LIN {X 0,Y 428.586,Z 1043.755,A -85,B 0,C 180,E1 19403.227,E2 19403.227} C_VEL
LIN {X 0,Y 431.846,Z 1036.608,A -85,B 0,C 180,E1 19403.942,E2 19403.942} C_VEL
LIN {X 0,Y 434.974,Z 1024.331,A -85,B 0,C 180,E1 19405.544,E2 19405.544} C_VEL
LIN {X 0,Y 437.859,Z 1011.623,A -85,B 0,C 180,E1 19407.088,E2 19407.088} C_VEL
LIN {X 0,Y 455.696,Z 965.576,A -85,B 0,C 180,E1 19410.268,E2 19410.268} C_VEL
LIN {X 0,Y 463.791,Z 940.685,A -85,B 0,C 180,E1 19411.605,E2 19411.605} C_VEL
LIN {X 0,Y 457.575,Z 919.275,A -85,B 0,C 180,E1 19415.61,E2 19415.61} C_VEL
LIN {X 0,Y 449.958,Z 899.264,A -85,B 0,C 180,E1 19420.368,E2 19420.368} C_VEL
LIN {X 0,Y 443.441,Z 884.682,A -85,B 0,C 180,E1 19425.003,E2 19425.003} C_VEL
LIN {X 0,Y 438.178,Z 874.111,A -85,B 0,C 180,E1 19429.684,E2 19429.684} C_VEL
LIN {X 0,Y 435.63,Z 868.79,A -85,B 0,C 180,E1 19433.016,E2 19433.016} C_VEL
LIN {X 0,Y 433.736,Z 862.951,A -85,B 0,C 180,E1 19438.99,E2 19438.99} C_VEL
LIN {X 0,Y 433.685,Z 863.847,A -85,B 0,C 180,E1 19442.859,E2 19442.859} C_VEL
LIN {X 0,Y 435.972,Z 870.801,A -85,B 0,C 180,E1 19448.898,E2 19448.898} C_VEL
LIN {X 0,Y 440.304,Z 880.375,A -85,B 0,C 180,E1 19453.887,E2 19453.887} C_VEL
LIN {X 0,Y 447.364,Z 897.231,A -85,B 0,C 180,E1 19459.727,E2 19459.727} C_VEL
LIN {X 0,Y 454.424,Z 917.787,A -85,B 0,C 180,E1 19464.863,E2 19464.863} C_VEL
LIN {X 0,Y 460.195,Z 940.594,A -85,B 0,C 180,E1 19469.353,E2 19469.353} C_VEL
LIN {X 0,Y 444.53,Z 983.942,A -85,B 0,C 180,E1 19472.239,E2 19472.239} C_VEL
LIN {X 0,Y 426.136,Z 1025.719,A -85,B 0,C 180,E1 19476.025,E2 19476.025} C_VEL
LIN {X 0,Y 408.075,Z 1061.829,A -85,B 0,C 180,E1 19480.461,E2 19480.461} C_VEL
LIN {X 0,Y 389.858,Z 1095.549,A -85,B 0,C 180,E1 19486.146,E2 19486.146} C_VEL
LIN {X 0,Y 374.87,Z 1122.588,A -85,B 0,C 180,E1 19492.358,E2 19492.358} C_VEL
LIN {X 0,Y 362.214,Z 1146.532,A -85,B 0,C 180,E1 19499.96,E2 19499.96} C_VEL
LIN {X 0,Y 354.663,Z 1163.186,A -85,B 0,C 180,E1 19507.453,E2 19507.453} C_VEL
LIN {X 0,Y 350.741,Z 1174.594,A -85,B 0,C 180,E1 19515.02,E2 19515.02} C_VEL
LIN {X 0,Y 349.218,Z 1181.313,A -85,B 0,C 180,E1 19522.542,E2 19522.542} C_VEL
LIN {X 0,Y 349.207,Z 1183.553,A -85,B 0,C 180,E1 19530.001,E2 19530.001} C_VEL
LIN {X 0,Y 349.289,Z 1181.244,A -85,B 0,C 180,E1 19537.459,E2 19537.459} C_VEL
LIN {X 0,Y 350.779,Z 1174.475,A -85,B 0,C 180,E1 19544.981,E2 19544.981} C_VEL
LIN {X 0,Y 354.739,Z 1163.013,A -85,B 0,C 180,E1 19552.545,E2 19552.545} C_VEL
LIN {X 0,Y 362.329,Z 1146.279,A -85,B 0,C 180,E1 19560.032,E2 19560.032} C_VEL
LIN {X 0,Y 375.056,Z 1122.213,A -85,B 0,C 180,E1 19567.648,E2 19567.648} C_VEL
LIN {X 0,Y 390.041,Z 1095.14,A -85,B 0,C 180,E1 19573.831,E2 19573.831} C_VEL
LIN {X 0,Y 408.55,Z 1060.855,A -85,B 0,C 180,E1 19579.582,E2 19579.582} C_VEL
LIN {X 0,Y 426.873,Z 1023.878,A -85,B 0,C 180,E1 19584.075,E2 19584.075} C_VEL
LIN {X 0,Y 444.921,Z 983.008,A -85,B 0,C 180,E1 19587.716,E2 19587.716} C_VEL
LIN {X 0,Y 460.201,Z 940.721,A -85,B 0,C 180,E1 19590.509,E2 19590.509} C_VEL
LIN {X 0,Y 454.389,Z 918.018,A -85,B 0,C 180,E1 19594.981,E2 19594.981} C_VEL
LIN {X 0,Y 447.112,Z 896.88,A -85,B 0,C 180,E1 19600.261,E2 19600.261} C_VEL
LIN {X 0,Y 440.513,Z 881.043,A -85,B 0,C 180,E1 19605.668,E2 19605.668} C_VEL
LIN {X 0,Y 436.198,Z 871.856,A -85,B 0,C 180,E1 19610.353,E2 19610.353} C_VEL
LIN {X 0,Y 434.863,Z 868.474,A -85,B 0,C 180,E1 19612.525,E2 19612.525} C_VEL
LIN {X 0,Y 433.446,Z 862.89,A -85,B 0,C 180,E1 19618.014,E2 19618.014} C_VEL
LIN {X 0,Y 433.74,Z 863.748,A -85,B 0,C 180,E1 19622.632,E2 19622.632} C_VEL
LIN {X 0,Y 436.694,Z 870.999,A -85,B 0,C 180,E1 19628.718,E2 19628.718} C_VEL
LIN {X 0,Y 441.953,Z 881.235,A -85,B 0,C 180,E1 19633.858,E2 19633.858} C_VEL
LIN {X 0,Y 449.143,Z 897.26,A -85,B 0,C 180,E1 19639.159,E2 19639.159} C_VEL
LIN {X 0,Y 457.134,Z 917.905,A -85,B 0,C 180,E1 19644.155,E2 19644.155} C_VEL
LIN {X 0,Y 463.866,Z 940.396,A -85,B 0,C 180,E1 19648.408,E2 19648.408} C_VEL
LIN {X 0,Y 449.596,Z 982.266,A -85,B 0,C 180,E1 19650.775,E2 19650.775} C_VEL
LIN {X 0,Y 431.875,Z 1025.293,A -85,B 0,C 180,E1 19654.114,E2 19654.114} C_VEL
LIN {X 0,Y 413.975,Z 1063.618,A -85,B 0,C 180,E1 19658.166,E2 19658.166} C_VEL
LIN {X 0,Y 395.325,Z 1100.234,A -85,B 0,C 180,E1 19663.486,E2 19663.486} C_VEL
LIN {X 0,Y 379.922,Z 1129.531,A -85,B 0,C 180,E1 19669.197,E2 19669.197} C_VEL
LIN {X 0,Y 366.111,Z 1156.35,A -85,B 0,C 180,E1 19676.315,E2 19676.315} C_VEL
LIN {X 0,Y 357.094,Z 1176.529,A -85,B 0,C 180,E1 19683.618,E2 19683.618} C_VEL
LIN {X 0,Y 351.628,Z 1191.995,A -85,B 0,C 180,E1 19691.651,E2 19691.651} C_VEL
LIN {X 0,Y 349.589,Z 1200.987,A -85,B 0,C 180,E1 19698.782,E2 19698.782} C_VEL
LIN {X 0,Y 349.086,Z 1205.302,A -85,B 0,C 180,E1 19705.032,E2 19705.032} C_VEL
LIN {X 0,Y 349.253,Z 1206.48,A -85,B 0,C 180,E1 19709.999,E2 19709.999} C_VEL
LIN {X 0,Y 349.173,Z 1204.011,A -85,B 0,C 180,E1 19717.459,E2 19717.459} C_VEL
LIN {X 0,Y 350.156,Z 1197.853,A -85,B 0,C 180,E1 19724.149,E2 19724.149} C_VEL
LIN {X 0,Y 353.578,Z 1185.77,A -85,B 0,C 180,E1 19731.958,E2 19731.958} C_VEL
LIN {X 0,Y 360.388,Z 1168.719,A -85,B 0,C 180,E1 19739.515,E2 19739.515} C_VEL
LIN {X 0,Y 372.131,Z 1144.328,A -85,B 0,C 180,E1 19747.157,E2 19747.157} C_VEL
LIN {X 0,Y 387.149,Z 1115.813,A -85,B 0,C 180,E1 19753.702,E2 19753.702} C_VEL
LIN {X 0,Y 405.824,Z 1080.003,A -85,B 0,C 180,E1 19759.666,E2 19759.666} C_VEL
LIN {X 0,Y 423.714,Z 1043.487,A -85,B 0,C 180,E1 19764.118,E2 19764.118} C_VEL
LIN {X 0,Y 437.859,Z 1011.623,A -85,B 0,C 180,E1 19767.088,E2 19767.088} C_VEL
LIN {X 0,Y 443.734,Z 986.824,A -85,B 0,C 180,E1 19769.787,E2 19769.787} C_VEL
LIN {X 0,Y 444.408,Z 984.999,A -85,B 0,C 180,E1 19769.923,E2 19769.923} C_VEL
LIN {X 0,Y 458.785,Z 943.642,A -85,B 0,C 180,E1 19772.398,E2 19772.398} C_VEL
LIN {X 0,Y 451.781,Z 920.233,A -85,B 0,C 180,E1 19777.109,E2 19777.109} C_VEL
LIN {X 0,Y 444.419,Z 900.847,A -85,B 0,C 180,E1 19782.183,E2 19782.183} C_VEL
LIN {X 0,Y 438.462,Z 887.226,A -85,B 0,C 180,E1 19787.045,E2 19787.045} C_VEL
LIN {X 0,Y 434.775,Z 879.627,A -85,B 0,C 180,E1 19790.991,E2 19790.991} C_VEL
LIN {X 0,Y 433.267,Z 876.2,A -85,B 0,C 180,E1 19793.229,E2 19793.229} C_VEL
LIN {X 0,Y 431.551,Z 870.535,A -85,B 0,C 180,E1 19798.985,E2 19798.985} C_VEL
LIN {X 0,Y 431.475,Z 871.393,A -85,B 0,C 180,E1 19802.748,E2 19802.748} C_VEL
LIN {X 0,Y 433.507,Z 877.891,A -85,B 0,C 180,E1 19808.536,E2 19808.536} C_VEL
LIN {X 0,Y 437.705,Z 888.299,A -85,B 0,C 180,E1 19813.971,E2 19813.971} C_VEL
LIN {X 0,Y 443.762,Z 903.724,A -85,B 0,C 180,E1 19819.376,E2 19819.376} C_VEL
LIN {X 0,Y 450.263,Z 923.937,A -85,B 0,C 180,E1 19824.524,E2 19824.524} C_VEL
LIN {X 0,Y 455.052,Z 944.062,A -85,B 0,C 180,E1 19828.604,E2 19828.604} C_VEL
LIN {X 0,Y 443.783,Z 975.55,A -85,B 0,C 180,E1 19830.729,E2 19830.729} C_VEL
LIN {X 0,Y 426.406,Z 1015.666,A -85,B 0,C 180,E1 19834.07,E2 19834.07} C_VEL
LIN {X 0,Y 407.054,Z 1054.1,A -85,B 0,C 180,E1 19838.476,E2 19838.476} C_VEL
LIN {X 0,Y 388.95,Z 1087.233,A -85,B 0,C 180,E1 19843.65,E2 19843.65} C_VEL
LIN {X 0,Y 372.018,Z 1116.573,A -85,B 0,C 180,E1 19849.952,E2 19849.952} C_VEL
LIN {X 0,Y 358.903,Z 1140.024,A -85,B 0,C 180,E1 19856.816,E2 19856.816} C_VEL
LIN {X 0,Y 348.66,Z 1159.953,A -85,B 0,C 180,E1 19865.102,E2 19865.102} C_VEL
LIN {X 0,Y 344.049,Z 1171.621,A -85,B 0,C 180,E1 19872.096,E2 19872.096} C_VEL
LIN {X 0,Y 341.71,Z 1179.921,A -85,B 0,C 180,E1 19879.813,E2 19879.813} C_VEL
LIN {X 0,Y 341.121,Z 1183.502,A -85,B 0,C 180,E1 19887.462,E2 19887.462} C_VEL
LIN {X 0,Y 341.232,Z 1183.485,A -85,B 0,C 180,E1 19892.539,E2 19892.539} C_VEL
LIN {X 0,Y 341.765,Z 1179.847,A -85,B 0,C 180,E1 19900.188,E2 19900.188} C_VEL
LIN {X 0,Y 344.103,Z 1171.477,A -85,B 0,C 180,E1 19907.904,E2 19907.904} C_VEL
LIN {X 0,Y 350.078,Z 1156.974,A -85,B 0,C 180,E1 19916.261,E2 19916.261} C_VEL
LIN {X 0,Y 359.934,Z 1137.868,A -85,B 0,C 180,E1 19923.8,E2 19923.8} C_VEL
LIN {X 0,Y 374.138,Z 1112.783,A -85,B 0,C 180,E1 19930.895,E2 19930.895} C_VEL
LIN {X 0,Y 390.81,Z 1083.708,A -85,B 0,C 180,E1 19936.873,E2 19936.873} C_VEL
LIN {X 0,Y 409.721,Z 1049.044,A -85,B 0,C 180,E1 19942.082,E2 19942.082} C_VEL
LIN {X 0,Y 427.732,Z 1012.531,A -85,B 0,C 180,E1 19946.123,E2 19946.123} C_VEL
LIN {X 0,Y 446.584,Z 968.32,A -85,B 0,C 180,E1 19949.677,E2 19949.677} C_VEL
LIN {X 0,Y 455.082,Z 944.515,A -85,B 0,C 180,E1 19951.205,E2 19951.205} C_VEL
LIN {X 0,Y 449.389,Z 921.401,A -85,B 0,C 180,E1 19955.954,E2 19955.954} C_VEL
LIN {X 0,Y 442.896,Z 901.812,A -85,B 0,C 180,E1 19961.102,E2 19961.102} C_VEL
LIN {X 0,Y 437.485,Z 887.883,A -85,B 0,C 180,E1 19966.022,E2 19966.022} C_VEL
LIN {X 0,Y 432.894,Z 876.3,A -85,B 0,C 180,E1 19972.202,E2 19972.202} C_VEL
LIN {X 0,Y 431.26,Z 870.482,A -85,B 0,C 180,E1 19978.004,E2 19978.004} C_VEL
LIN {X 0,Y 431.52,Z 871.282,A -85,B 0,C 180,E1 19982.52,E2 19982.52} C_VEL
LIN {X 0,Y 434.321,Z 878.522,A -85,B 0,C 180,E1 19988.575,E2 19988.575} C_VEL
LIN {X 0,Y 438.944,Z 887.899,A -85,B 0,C 180,E1 19993.447,E2 19993.447} C_VEL
LIN {X 0,Y 445.778,Z 903.809,A -85,B 0,C 180,E1 19998.795,E2 19998.795} C_VEL
LIN {X 0,Y 453.312,Z 924.562,A -85,B 0,C 180,E1 20003.896,E2 20003.896} C_VEL
LIN {X 0,Y 458.761,Z 943.784,A -85,B 0,C 180,E1 20007.646,E2 20007.646} C_VEL
LIN {X 0,Y 442.236,Z 990.175,A -85,B 0,C 180,E1 20010.438,E2 20010.438} C_VEL
LIN {X 0,Y 424.86,Z 1030.734,A -85,B 0,C 180,E1 20013.733,E2 20013.733} C_VEL
LIN {X 0,Y 405.075,Z 1070.686,A -85,B 0,C 180,E1 20018.2,E2 20018.2} C_VEL
LIN {X 0,Y 386.799,Z 1105.278,A -85,B 0,C 180,E1 20023.515,E2 20023.515} C_VEL
LIN {X 0,Y 369.335,Z 1137.111,A -85,B 0,C 180,E1 20030.255,E2 20030.255} C_VEL
LIN {X 0,Y 356.233,Z 1162.098,A -85,B 0,C 180,E1 20037.567,E2 20037.567} C_VEL
LIN {X 0,Y 347.526,Z 1181.212,A -85,B 0,C 180,E1 20045.333,E2 20045.333} C_VEL
LIN {X 0,Y 343.523,Z 1193.016,A -85,B 0,C 180,E1 20052.065,E2 20052.065} C_VEL
LIN {X 0,Y 341.538,Z 1201.955,A -85,B 0,C 180,E1 20059.805,E2 20059.805} C_VEL
LIN {X 0,Y 341.228,Z 1205.87,A -85,B 0,C 180,E1 20067.461,E2 20067.461} C_VEL
LIN {X 0,Y 341.323,Z 1205.874,A -85,B 0,C 180,E1 20072.536,E2 20072.536} C_VEL
LIN {X 0,Y 341.534,Z 1201.962,A -85,B 0,C 180,E1 20080.193,E2 20080.193} C_VEL
LIN {X 0,Y 343.512,Z 1193.03,A -85,B 0,C 180,E1 20087.933,E2 20087.933} C_VEL
LIN {X 0,Y 348.459,Z 1179.029,A -85,B 0,C 180,E1 20095.698,E2 20095.698} C_VEL
LIN {X 0,Y 357.511,Z 1159.576,A -85,B 0,C 180,E1 20103.33,E2 20103.33} C_VEL
LIN {X 0,Y 371.226,Z 1133.502,A -85,B 0,C 180,E1 20110.638,E2 20110.638} C_VEL
LIN {X 0,Y 388.234,Z 1102.606,A -85,B 0,C 180,E1 20116.975,E2 20116.975} C_VEL
LIN {X 0,Y 408.129,Z 1064.976,A -85,B 0,C 180,E1 20122.545,E2 20122.545} C_VEL
LIN {X 0,Y 426.367,Z 1027.477,A -85,B 0,C 180,E1 20126.576,E2 20126.576} C_VEL
LIN {X 0,Y 444.095,Z 985.792,A -85,B 0,C 180,E1 20129.867,E2 20129.867} C_VEL
LIN {X 0,Y 444.408,Z 984.999,A -85,B 0,C 180,E1 20129.923,E2 20129.923} C_VEL
LIN {X 0,Y 447.634,Z 971.252,A -85,B 0,C 180,E1 20131.267,E2 20131.267} C_VEL
LIN {X 0,Y 450.696,Z 957.074,A -85,B 0,C 180,E1 20132.515,E2 20132.515} C_VEL
LIN {X 0,Y 453.804,Z 947.912,A -85,B 0,C 180,E1 20133.003,E2 20133.003} C_VEL
LIN {X 0,Y 447.279,Z 924.708,A -85,B 0,C 180,E1 20137.868,E2 20137.868} C_VEL
LIN {X 0,Y 440.411,Z 905.787,A -85,B 0,C 180,E1 20143.033,E2 20143.033} C_VEL
LIN {X 0,Y 434.032,Z 890.643,A -85,B 0,C 180,E1 20148.95,E2 20148.95} C_VEL
LIN {X 0,Y 430.496,Z 883.205,A -85,B 0,C 180,E1 20153.944,E2 20153.944} C_VEL
LIN {X 0,Y 429.364,Z 878.125,A -85,B 0,C 180,E1 20158.98,E2 20158.98} C_VEL
LIN {X 0,Y 429.347,Z 878.148,A -85,B 0,C 180,E1 20162.005,E2 20162.005} C_VEL
LIN {X 0,Y 430.92,Z 885.665,A -85,B 0,C 180,E1 20168.588,E2 20168.588} C_VEL
LIN {X 0,Y 435.081,Z 896.244,A -85,B 0,C 180,E1 20174.057,E2 20174.057} C_VEL
LIN {X 0,Y 440.747,Z 911.938,A -85,B 0,C 180,E1 20179.514,E2 20179.514} C_VEL
LIN {X 0,Y 446.572,Z 932.006,A -85,B 0,C 180,E1 20184.606,E2 20184.606} C_VEL
LIN {X 0,Y 450.102,Z 948.566,A -85,B 0,C 180,E1 20188.019,E2 20188.019} C_VEL
LIN {X 0,Y 431.793,Z 994.267,A -85,B 0,C 180,E1 20191.22,E2 20191.22} C_VEL
LIN {X 0,Y 413.229,Z 1033.294,A -85,B 0,C 180,E1 20194.973,E2 20194.973} C_VEL
LIN {X 0,Y 393.426,Z 1069.906,A -85,B 0,C 180,E1 20199.811,E2 20199.811} C_VEL
LIN {X 0,Y 375.588,Z 1100.457,A -85,B 0,C 180,E1 20205.308,E2 20205.308} C_VEL
LIN {X 0,Y 358.669,Z 1128.649,A -85,B 0,C 180,E1 20212.347,E2 20212.347} C_VEL
LIN {X 0,Y 347.218,Z 1148.728,A -85,B 0,C 180,E1 20219.247,E2 20219.247} C_VEL
LIN {X 0,Y 339.184,Z 1164.828,A -85,B 0,C 180,E1 20227.058,E2 20227.058} C_VEL
LIN {X 0,Y 335.205,Z 1175.121,A -85,B 0,C 180,E1 20234.308,E2 20234.308} C_VEL
LIN {X 0,Y 333.46,Z 1181.833,A -85,B 0,C 180,E1 20242.188,E2 20242.188} C_VEL
LIN {X 0,Y 333.411,Z 1184.071,A -85,B 0,C 180,E1 20250.001,E2 20250.001} C_VEL
LIN {X 0,Y 333.521,Z 1181.766,A -85,B 0,C 180,E1 20257.813,E2 20257.813} C_VEL
LIN {X 0,Y 335.256,Z 1175.005,A -85,B 0,C 180,E1 20265.692,E2 20265.692} C_VEL
LIN {X 0,Y 340.463,Z 1162.3,A -85,B 0,C 180,E1 20274.31,E2 20274.31} C_VEL
LIN {X 0,Y 350.146,Z 1143.453,A -85,B 0,C 180,E1 20282.641,E2 20282.641} C_VEL
LIN {X 0,Y 363.929,Z 1119.888,A -85,B 0,C 180,E1 20290.007,E2 20290.007} C_VEL
LIN {X 0,Y 381.77,Z 1089.961,A -85,B 0,C 180,E1 20296.663,E2 20296.663} C_VEL
LIN {X 0,Y 400.454,Z 1057.184,A -85,B 0,C 180,E1 20301.952,E2 20301.952} C_VEL
LIN {X 0,Y 420.938,Z 1017.603,A -85,B 0,C 180,E1 20306.581,E2 20306.581} C_VEL
LIN {X 0,Y 439.163,Z 977.032,A -85,B 0,C 180,E1 20309.977,E2 20309.977} C_VEL
LIN {X 0,Y 449.962,Z 948.025,A -85,B 0,C 180,E1 20311.972,E2 20311.972} C_VEL
LIN {X 0,Y 444.767,Z 925.808,A -85,B 0,C 180,E1 20316.718,E2 20316.718} C_VEL
LIN {X 0,Y 438.761,Z 906.785,A -85,B 0,C 180,E1 20321.957,E2 20321.957} C_VEL
LIN {X 0,Y 433.906,Z 893.651,A -85,B 0,C 180,E1 20326.931,E2 20326.931} C_VEL
LIN {X 0,Y 430.008,Z 883.44,A -85,B 0,C 180,E1 20332.812,E2 20332.812} C_VEL
LIN {X 0,Y 429.073,Z 878.075,A -85,B 0,C 180,E1 20337.994,E2 20337.994} C_VEL
LIN {X 0,Y 429.294,Z 879.012,A -85,B 0,C 180,E1 20342.533,E2 20342.533} C_VEL
LIN {X 0,Y 432.017,Z 886.651,A -85,B 0,C 180,E1 20348.81,E2 20348.81} C_VEL
LIN {X 0,Y 436.314,Z 895.901,A -85,B 0,C 180,E1 20353.53,E2 20353.53} C_VEL
LIN {X 0,Y 442.771,Z 912.014,A -85,B 0,C 180,E1 20358.928,E2 20358.928} C_VEL
LIN {X 0,Y 449.428,Z 931.869,A -85,B 0,C 180,E1 20363.805,E2 20363.805} C_VEL
LIN {X 0,Y 453.692,Z 947.9,A -85,B 0,C 180,E1 20367.002,E2 20367.002} C_VEL
LIN {X 0,Y 436.967,Z 992.903,A -85,B 0,C 180,E1 20369.729,E2 20369.729} C_VEL
LIN {X 0,Y 419.212,Z 1032.761,A -85,B 0,C 180,E1 20373.026,E2 20373.026} C_VEL
LIN {X 0,Y 398.464,Z 1073.371,A -85,B 0,C 180,E1 20377.658,E2 20377.658} C_VEL
LIN {X 0,Y 379.725,Z 1107.337,A -85,B 0,C 180,E1 20383.042,E2 20383.042} C_VEL
LIN {X 0,Y 362.274,Z 1138.074,A -85,B 0,C 180,E1 20389.718,E2 20389.718} C_VEL
LIN {X 0,Y 348.73,Z 1162.77,A -85,B 0,C 180,E1 20397.174,E2 20397.174} C_VEL
LIN {X 0,Y 339.719,Z 1181.772,A -85,B 0,C 180,E1 20405.153,E2 20405.153} C_VEL
LIN {X 0,Y 335.255,Z 1194.611,A -85,B 0,C 180,E1 20412.962,E2 20412.962} C_VEL
LIN {X 0,Y 333.664,Z 1201.692,A -85,B 0,C 180,E1 20419.562,E2 20419.562} C_VEL
LIN {X 0,Y 333.322,Z 1205.61,A -85,B 0,C 180,E1 20427.4,E2 20427.4} C_VEL
LIN {X 0,Y 333.413,Z 1205.614,A -85,B 0,C 180,E1 20432.596,E2 20432.596} C_VEL
LIN {X 0,Y 333.659,Z 1201.7,A -85,B 0,C 180,E1 20440.436,E2 20440.436} C_VEL
LIN {X 0,Y 335.787,Z 1192.764,A -85,B 0,C 180,E1 20448.36,E2 20448.36} C_VEL
LIN {X 0,Y 341.553,Z 1177.754,A -85,B 0,C 180,E1 20456.777,E2 20456.777} C_VEL
LIN {X 0,Y 351.226,Z 1158.109,A -85,B 0,C 180,E1 20464.458,E2 20464.458} C_VEL
LIN {X 0,Y 366.464,Z 1130.803,A -85,B 0,C 180,E1 20472.066,E2 20472.066} C_VEL
LIN {X 0,Y 383.468,Z 1100.772,A -85,B 0,C 180,E1 20478.15,E2 20478.15} C_VEL
LIN {X 0,Y 403.874,Z 1063.446,A -85,B 0,C 180,E1 20483.633,E2 20483.633} C_VEL
LIN {X 0,Y 422.597,Z 1025.656,A -85,B 0,C 180,E1 20487.65,E2 20487.65} C_VEL
LIN {X 0,Y 441.25,Z 982.609,A -85,B 0,C 180,E1 20490.984,E2 20490.984} C_VEL
LIN {X 0,Y 450.696,Z 957.074,A -85,B 0,C 180,E1 20492.515,E2 20492.515} C_VEL
LIN {X 0,Y 451.033,Z 951.97,A -85,B 0,C 180,E1 20493.12,E2 20493.12} C_VEL
LIN {X 0,Y 447.15,Z 945.009,A -85,B 0,C 180,E1 20495.079,E2 20495.079} C_VEL
LIN {X 0,Y 440.482,Z 922.195,A -85,B 0,C 180,E1 20500.449,E2 20500.449} C_VEL
LIN {X 0,Y 434.204,Z 905.416,A -85,B 0,C 180,E1 20505.89,E2 20505.89} C_VEL
LIN {X 0,Y 429.736,Z 894.929,A -85,B 0,C 180,E1 20510.938,E2 20510.938} C_VEL
LIN {X 0,Y 427.973,Z 890.717,A -85,B 0,C 180,E1 20513.908,E2 20513.908} C_VEL
LIN {X 0,Y 426.946,Z 886.447,A -85,B 0,C 180,E1 20517.96,E2 20517.96} C_VEL
LIN {X 0,Y 426.854,Z 885.745,A -85,B 0,C 180,E1 20522.017,E2 20522.017} C_VEL
LIN {X 0,Y 428.64,Z 894.364,A -85,B 0,C 180,E1 20529.219,E2 20529.219} C_VEL
LIN {X 0,Y 432.567,Z 905.279,A -85,B 0,C 180,E1 20534.657,E2 20534.657} C_VEL
LIN {X 0,Y 437.431,Z 919.79,A -85,B 0,C 180,E1 20539.617,E2 20539.617} C_VEL
LIN {X 0,Y 442.63,Z 939.883,A -85,B 0,C 180,E1 20544.706,E2 20544.706} C_VEL
LIN {X 0,Y 444.75,Z 953.456,A -85,B 0,C 180,E1 20547.43,E2 20547.43} C_VEL
LIN {X 0,Y 426.466,Z 997.264,A -85,B 0,C 180,E1 20550.52,E2 20550.52} C_VEL
LIN {X 0,Y 407.51,Z 1035.613,A -85,B 0,C 180,E1 20554.277,E2 20554.277} C_VEL
LIN {X 0,Y 387.266,Z 1071.894,A -85,B 0,C 180,E1 20559.149,E2 20559.149} C_VEL
LIN {X 0,Y 368.683,Z 1102.47,A -85,B 0,C 180,E1 20564.799,E2 20564.799} C_VEL
LIN {X 0,Y 351.557,Z 1129.978,A -85,B 0,C 180,E1 20571.84,E2 20571.84} C_VEL
LIN {X 0,Y 339.307,Z 1150.484,A -85,B 0,C 180,E1 20579.194,E2 20579.194} C_VEL
LIN {X 0,Y 330.695,Z 1167.316,A -85,B 0,C 180,E1 20587.854,E2 20587.854} C_VEL
LIN {X 0,Y 326.738,Z 1177.715,A -85,B 0,C 180,E1 20596.126,E2 20596.126} C_VEL
LIN {X 0,Y 325.575,Z 1182.094,A -85,B 0,C 180,E1 20601.997,E2 20601.997} C_VEL
LIN {X 0,Y 325.519,Z 1184.33,A -85,B 0,C 180,E1 20610.001,E2 20610.001} C_VEL
LIN {X 0,Y 325.635,Z 1182.028,A -85,B 0,C 180,E1 20618.004,E2 20618.004} C_VEL
LIN {X 0,Y 327.525,Z 1175.27,A -85,B 0,C 180,E1 20626.072,E2 20626.072} C_VEL
LIN {X 0,Y 333.072,Z 1162.532,A -85,B 0,C 180,E1 20634.906,E2 20634.906} C_VEL
LIN {X 0,Y 342.939,Z 1144.227,A -85,B 0,C 180,E1 20643.191,E2 20643.191} C_VEL
LIN {X 0,Y 357.042,Z 1121.216,A -85,B 0,C 180,E1 20650.581,E2 20650.581} C_VEL
LIN {X 0,Y 375.295,Z 1091.664,A -85,B 0,C 180,E1 20657.294,E2 20657.294} C_VEL
LIN {X 0,Y 394.308,Z 1059.607,A -85,B 0,C 180,E1 20662.59,E2 20662.59} C_VEL
LIN {X 0,Y 415.317,Z 1020.201,A -85,B 0,C 180,E1 20667.278,E2 20667.278} C_VEL
LIN {X 0,Y 433.574,Z 981.244,A -85,B 0,C 180,E1 20670.613,E2 20670.613} C_VEL
LIN {X 0,Y 444.833,Z 952.026,A -85,B 0,C 180,E1 20672.65,E2 20672.65} C_VEL
LIN {X 0,Y 440.425,Z 931.006,A -85,B 0,C 180,E1 20677.31,E2 20677.31} C_VEL
LIN {X 0,Y 435.251,Z 913.259,A -85,B 0,C 180,E1 20682.329,E2 20682.329} C_VEL
LIN {X 0,Y 430.644,Z 900.17,A -85,B 0,C 180,E1 20687.426,E2 20687.426} C_VEL
LIN {X 0,Y 427.434,Z 891.066,A -85,B 0,C 180,E1 20692.787,E2 20692.787} C_VEL
LIN {X 0,Y 426.612,Z 885.588,A -85,B 0,C 180,E1 20697.982,E2 20697.982} C_VEL
LIN {X 0,Y 426.841,Z 885.953,A -85,B 0,C 180,E1 20702.04,E2 20702.04} C_VEL
LIN {X 0,Y 429.445,Z 894.352,A -85,B 0,C 180,E1 20708.863,E2 20708.863} C_VEL
LIN {X 0,Y 434.118,Z 905.122,A -85,B 0,C 180,E1 20714.113,E2 20714.113} C_VEL
LIN {X 0,Y 439.785,Z 920.128,A -85,B 0,C 180,E1 20719.061,E2 20719.061} C_VEL
LIN {X 0,Y 446.398,Z 941.96,A -85,B 0,C 180,E1 20724.325,E2 20724.325} C_VEL
LIN {X 0,Y 448.256,Z 952.932,A -85,B 0,C 180,E1 20726.369,E2 20726.369} C_VEL
LIN {X 0,Y 431.254,Z 996.887,A -85,B 0,C 180,E1 20729.091,E2 20729.091} C_VEL
LIN {X 0,Y 412.372,Z 1037.308,A -85,B 0,C 180,E1 20732.559,E2 20732.559} C_VEL
LIN {X 0,Y 392.434,Z 1075.038,A -85,B 0,C 180,E1 20736.963,E2 20736.963} C_VEL
LIN {X 0,Y 372.648,Z 1109.454,A -85,B 0,C 180,E1 20742.562,E2 20742.562} C_VEL
LIN {X 0,Y 355.249,Z 1139.02,A -85,B 0,C 180,E1 20749.154,E2 20749.154} C_VEL
LIN {X 0,Y 340.813,Z 1164.345,A -85,B 0,C 180,E1 20757.102,E2 20757.102} C_VEL
LIN {X 0,Y 331.839,Z 1182.568,A -85,B 0,C 180,E1 20765.087,E2 20765.087} C_VEL
LIN {X 0,Y 327.516,Z 1194.344,A -85,B 0,C 180,E1 20772.547,E2 20772.547} C_VEL
LIN {X 0,Y 325.79,Z 1201.429,A -85,B 0,C 180,E1 20779.307,E2 20779.307} C_VEL
LIN {X 0,Y 325.426,Z 1205.35,A -85,B 0,C 180,E1 20787.337,E2 20787.337} C_VEL
LIN {X 0,Y 325.511,Z 1205.354,A -85,B 0,C 180,E1 20792.659,E2 20792.659} C_VEL
LIN {X 0,Y 325.785,Z 1201.437,A -85,B 0,C 180,E1 20800.691,E2 20800.691} C_VEL
LIN {X 0,Y 328.099,Z 1192.498,A -85,B 0,C 180,E1 20808.806,E2 20808.806} C_VEL
LIN {X 0,Y 333.703,Z 1178.491,A -85,B 0,C 180,E1 20816.924,E2 20816.924} C_VEL
LIN {X 0,Y 343.752,Z 1159.033,A -85,B 0,C 180,E1 20824.851,E2 20824.851} C_VEL
LIN {X 0,Y 358.816,Z 1132.962,A -85,B 0,C 180,E1 20832.361,E2 20832.361} C_VEL
LIN {X 0,Y 376.705,Z 1102.785,A -85,B 0,C 180,E1 20838.695,E2 20838.695} C_VEL
LIN {X 0,Y 397.245,Z 1066.363,A -85,B 0,C 180,E1 20844.181,E2 20844.181} C_VEL
LIN {X 0,Y 416.934,Z 1028.278,A -85,B 0,C 180,E1 20848.335,E2 20848.335} C_VEL
LIN {X 0,Y 435.41,Z 987.091,A -85,B 0,C 180,E1 20851.589,E2 20851.589} C_VEL
LIN {X 0,Y 448.667,Z 951.554,A -85,B 0,C 180,E1 20853.757,E2 20853.757} C_VEL
LIN {X 0,Y 447.15,Z 945.009,A -85,B 0,C 180,E1 20855.079,E2 20855.079} C_VEL
LIN {X 0,Y 444.07,Z 940.362,A -85,B 0,C 180,E1 20856.608,E2 20856.608} C_VEL
LIN {X 0,Y 438.265,Z 934.315,A -85,B 0,C 180,E1 20859.267,E2 20859.267} C_VEL
LIN {X 0,Y 432.781,Z 917.31,A -85,B 0,C 180,E1 20864.29,E2 20864.29} C_VEL
LIN {X 0,Y 427.921,Z 904.246,A -85,B 0,C 180,E1 20869.82,E2 20869.82} C_VEL
LIN {X 0,Y 425.222,Z 897.881,A -85,B 0,C 180,E1 20874.278,E2 20874.278} C_VEL
LIN {X 0,Y 424.295,Z 893.014,A -85,B 0,C 180,E1 20879.988,E2 20879.988} C_VEL
LIN {X 0,Y 424.286,Z 893.349,A -85,B 0,C 180,E1 20882.029,E2 20882.029} C_VEL
LIN {X 0,Y 425.866,Z 901.944,A -85,B 0,C 180,E1 20889.28,E2 20889.28} C_VEL
LIN {X 0,Y 430.087,Z 914.336,A -85,B 0,C 180,E1 20895.265,E2 20895.265} C_VEL
LIN {X 0,Y 434.587,Z 929.905,A -85,B 0,C 180,E1 20900.332,E2 20900.332} C_VEL
LIN {X 0,Y 438.947,Z 949.77,A -85,B 0,C 180,E1 20905.218,E2 20905.218} C_VEL
LIN {X 0,Y 439.821,Z 957.051,A -85,B 0,C 180,E1 20906.712,E2 20906.712} C_VEL
LIN {X 0,Y 421.189,Z 1000.25,A -85,B 0,C 180,E1 20909.8,E2 20909.8} C_VEL
LIN {X 0,Y 400.394,Z 1040.59,A -85,B 0,C 180,E1 20913.873,E2 20913.873} C_VEL
LIN {X 0,Y 380.148,Z 1075.511,A -85,B 0,C 180,E1 20918.732,E2 20918.732} C_VEL
LIN {X 0,Y 360.882,Z 1105.988,A -85,B 0,C 180,E1 20924.617,E2 20924.617} C_VEL
LIN {X 0,Y 344.473,Z 1131.307,A -85,B 0,C 180,E1 20931.311,E2 20931.311} C_VEL
LIN {X 0,Y 331.39,Z 1152.242,A -85,B 0,C 180,E1 20939.138,E2 20939.138} C_VEL
LIN {X 0,Y 322.694,Z 1168.688,A -85,B 0,C 180,E1 20948,E2 20948} C_VEL
LIN {X 0,Y 318.803,Z 1178.407,A -85,B 0,C 180,E1 20956.292,E2 20956.292} C_VEL
LIN {X 0,Y 317.482,Z 1183.535,A -85,B 0,C 180,E1 20964.539,E2 20964.539} C_VEL
LIN {X 0,Y 317.619,Z 1184.59,A -85,B 0,C 180,E1 20970.001,E2 20970.001} C_VEL
LIN {X 0,Y 317.775,Z 1182.289,A -85,B 0,C 180,E1 20978.203,E2 20978.203} C_VEL
LIN {X 0,Y 319.782,Z 1175.535,A -85,B 0,C 180,E1 20986.472,E2 20986.472} C_VEL
LIN {X 0,Y 325.676,Z 1162.802,A -85,B 0,C 180,E1 20995.512,E2 20995.512} C_VEL
LIN {X 0,Y 336.079,Z 1144.499,A -85,B 0,C 180,E1 21003.96,E2 21003.96} C_VEL
LIN {X 0,Y 350.861,Z 1121.48,A -85,B 0,C 180,E1 21011.454,E2 21011.454} C_VEL
LIN {X 0,Y 369.766,Z 1091.936,A -85,B 0,C 180,E1 21018.231,E2 21018.231} C_VEL
LIN {X 0,Y 389.726,Z 1059.306,A -85,B 0,C 180,E1 21023.622,E2 21023.622} C_VEL
LIN {X 0,Y 411.506,Z 1019.519,A -85,B 0,C 180,E1 21028.322,E2 21028.322} C_VEL
LIN {X 0,Y 430.687,Z 979.103,A -85,B 0,C 180,E1 21031.721,E2 21031.721} C_VEL
LIN {X 0,Y 439.818,Z 956.235,A -85,B 0,C 180,E1 21033.293,E2 21033.293} C_VEL
LIN {X 0,Y 435.834,Z 935.705,A -85,B 0,C 180,E1 21038.011,E2 21038.011} C_VEL
LIN {X 0,Y 431.146,Z 918.339,A -85,B 0,C 180,E1 21043.139,E2 21043.139} C_VEL
LIN {X 0,Y 426.798,Z 904.82,A -85,B 0,C 180,E1 21048.784,E2 21048.784} C_VEL
LIN {X 0,Y 424.85,Z 898.57,A -85,B 0,C 180,E1 21052.765,E2 21052.765} C_VEL
LIN {X 0,Y 424.066,Z 893.124,A -85,B 0,C 180,E1 21057.97,E2 21057.97} C_VEL
LIN {X 0,Y 424.276,Z 893.547,A -85,B 0,C 180,E1 21062.053,E2 21062.053} C_VEL
LIN {X 0,Y 426.862,Z 902.014,A -85,B 0,C 180,E1 21068.917,E2 21068.917} C_VEL
LIN {X 0,Y 431.186,Z 912.891,A -85,B 0,C 180,E1 21074.211,E2 21074.211} C_VEL
LIN {X 0,Y 436.788,Z 929.245,A -85,B 0,C 180,E1 21079.466,E2 21079.466} C_VEL
LIN {X 0,Y 442.657,Z 951.124,A -85,B 0,C 180,E1 21084.663,E2 21084.663} C_VEL
LIN {X 0,Y 443.563,Z 955.611,A -85,B 0,C 180,E1 21085.56,E2 21085.56} C_VEL
LIN {X 0,Y 426.067,Z 999.41,A -85,B 0,C 180,E1 21088.346,E2 21088.346} C_VEL
LIN {X 0,Y 406.244,Z 1040.523,A -85,B 0,C 180,E1 21091.943,E2 21091.943} C_VEL
LIN {X 0,Y 385.928,Z 1077.553,A -85,B 0,C 180,E1 21096.381,E2 21096.381} C_VEL
LIN {X 0,Y 364.769,Z 1112.996,A -85,B 0,C 180,E1 21102.345,E2 21102.345} C_VEL
LIN {X 0,Y 347.565,Z 1141.021,A -85,B 0,C 180,E1 21108.898,E2 21108.898} C_VEL
LIN {X 0,Y 332.911,Z 1165.845,A -85,B 0,C 180,E1 21116.995,E2 21116.995} C_VEL
LIN {X 0,Y 323.811,Z 1183.485,A -85,B 0,C 180,E1 21125.164,E2 21125.164} C_VEL
LIN {X 0,Y 319.235,Z 1195.696,A -85,B 0,C 180,E1 21133.499,E2 21133.499} C_VEL
LIN {X 0,Y 317.943,Z 1201.166,A -85,B 0,C 180,E1 21139.039,E2 21139.039} C_VEL
LIN {X 0,Y 317.529,Z 1205.091,A -85,B 0,C 180,E1 21147.271,E2 21147.271} C_VEL
LIN {X 0,Y 317.614,Z 1205.095,A -85,B 0,C 180,E1 21152.726,E2 21152.726} C_VEL
LIN {X 0,Y 317.937,Z 1201.175,A -85,B 0,C 180,E1 21160.958,E2 21160.958} C_VEL
LIN {X 0,Y 320.439,Z 1192.075,A -85,B 0,C 180,E1 21169.386,E2 21169.386} C_VEL
LIN {X 0,Y 327,Z 1177.01,A -85,B 0,C 180,E1 21178.182,E2 21178.182} C_VEL
LIN {X 0,Y 337.756,Z 1157.472,A -85,B 0,C 180,E1 21186.08,E2 21186.08} C_VEL
LIN {X 0,Y 354.229,Z 1130.244,A -85,B 0,C 180,E1 21193.883,E2 21193.883} C_VEL
LIN {X 0,Y 372.711,Z 1100.043,A -85,B 0,C 180,E1 21200.084,E2 21200.084} C_VEL
LIN {X 0,Y 394.088,Z 1063.25,A -85,B 0,C 180,E1 21205.526,E2 21205.526} C_VEL
LIN {X 0,Y 413.982,Z 1025.314,A -85,B 0,C 180,E1 21209.546,E2 21209.546} C_VEL
LIN {X 0,Y 433.181,Z 983.083,A -85,B 0,C 180,E1 21212.794,E2 21212.794} C_VEL
LIN {X 0,Y 443.674,Z 955.679,A -85,B 0,C 180,E1 21214.441,E2 21214.441} C_VEL
LIN {X 0,Y 438.265,Z 934.315,A -85,B 0,C 180,E1 21219.267,E2 21219.267} C_VEL
LIN {X 0,Y 435.316,Z 930.715,A -85,B 0,C 180,E1 21220.879,E2 21220.879} C_VEL
LIN {X 0,Y 430.114,Z 926.675,A -85,B 0,C 180,E1 21223.678,E2 21223.678} C_VEL
LIN {X 0,Y 425.353,Z 912.869,A -85,B 0,C 180,E1 21229.24,E2 21229.24} C_VEL
LIN {X 0,Y 422.682,Z 905.722,A -85,B 0,C 180,E1 21233.832,E2 21233.832} C_VEL
LIN {X 0,Y 421.708,Z 900.496,A -85,B 0,C 180,E1 21239.988,E2 21239.988} C_VEL
LIN {X 0,Y 421.383,Z 902.247,A -85,B 0,C 180,E1 21243.174,E2 21243.174} C_VEL
LIN {X 0,Y 422.923,Z 909.307,A -85,B 0,C 180,E1 21249.239,E2 21249.239} C_VEL
LIN {X 0,Y 426.419,Z 920.781,A -85,B 0,C 180,E1 21254.873,E2 21254.873} C_VEL
LIN {X 0,Y 430.703,Z 936.971,A -85,B 0,C 180,E1 21260.229,E2 21260.229} C_VEL
LIN {X 0,Y 434.52,Z 957.439,A -85,B 0,C 180,E1 21265.288,E2 21265.288} C_VEL
LIN {X 0,Y 434.581,Z 961.593,A -85,B 0,C 180,E1 21266.035,E2 21266.035} C_VEL
LIN {X 0,Y 415.946,Z 1003.047,A -85,B 0,C 180,E1 21269.061,E2 21269.061} C_VEL
LIN {X 0,Y 394.008,Z 1044.305,A -85,B 0,C 180,E1 21273.307,E2 21273.307} C_VEL
LIN {X 0,Y 373.008,Z 1078.922,A -85,B 0,C 180,E1 21278.29,E2 21278.29} C_VEL
LIN {X 0,Y 352.113,Z 1110.819,A -85,B 0,C 180,E1 21284.707,E2 21284.707} C_VEL
LIN {X 0,Y 334.77,Z 1136.423,A -85,B 0,C 180,E1 21292.075,E2 21292.075} C_VEL
LIN {X 0,Y 322.328,Z 1156.006,A -85,B 0,C 180,E1 21300.007,E2 21300.007} C_VEL
LIN {X 0,Y 314.488,Z 1170.303,A -85,B 0,C 180,E1 21308.466,E2 21308.466} C_VEL
LIN {X 0,Y 310.916,Z 1178.98,A -85,B 0,C 180,E1 21316.321,E2 21316.321} C_VEL
LIN {X 0,Y 309.584,Z 1183.795,A -85,B 0,C 180,E1 21324.399,E2 21324.399} C_VEL
LIN {X 0,Y 309.731,Z 1184.849,A -85,B 0,C 180,E1 21330.001,E2 21330.001} C_VEL
LIN {X 0,Y 309.893,Z 1182.551,A -85,B 0,C 180,E1 21338.413,E2 21338.413} C_VEL
LIN {X 0,Y 312.082,Z 1175.8,A -85,B 0,C 180,E1 21346.891,E2 21346.891} C_VEL
LIN {X 0,Y 318.241,Z 1163.231,A -85,B 0,C 180,E1 21356.056,E2 21356.056} C_VEL
LIN {X 0,Y 329.788,Z 1143.96,A -85,B 0,C 180,E1 21365.083,E2 21365.083} C_VEL
LIN {X 0,Y 345.502,Z 1120.537,A -85,B 0,C 180,E1 21372.683,E2 21372.683} C_VEL
LIN {X 0,Y 365.981,Z 1089.706,A -85,B 0,C 180,E1 21379.693,E2 21379.693} C_VEL
LIN {X 0,Y 387.042,Z 1056.012,A -85,B 0,C 180,E1 21385.076,E2 21385.076} C_VEL
LIN {X 0,Y 407.645,Z 1019.259,A -85,B 0,C 180,E1 21389.333,E2 21389.333} C_VEL
LIN {X 0,Y 427.081,Z 979.055,A -85,B 0,C 180,E1 21392.691,E2 21392.691} C_VEL
LIN {X 0,Y 434.828,Z 960.244,A -85,B 0,C 180,E1 21393.994,E2 21393.994} C_VEL
LIN {X 0,Y 431.522,Z 941.479,A -85,B 0,C 180,E1 21398.442,E2 21398.442} C_VEL
LIN {X 0,Y 427.347,Z 924.562,A -85,B 0,C 180,E1 21403.582,E2 21403.582} C_VEL
LIN {X 0,Y 423.851,Z 912.54,A -85,B 0,C 180,E1 21408.705,E2 21408.705} C_VEL
LIN {X 0,Y 421.526,Z 904.955,A -85,B 0,C 180,E1 21413.839,E2 21413.839} C_VEL
LIN {X 0,Y 421.428,Z 900.662,A -85,B 0,C 180,E1 21417.957,E2 21417.957} C_VEL
LIN {X 0,Y 421.657,Z 901.113,A -85,B 0,C 180,E1 21422.065,E2 21422.065} C_VEL
LIN {X 0,Y 423.55,Z 908.245,A -85,B 0,C 180,E1 21428.216,E2 21428.216} C_VEL
LIN {X 0,Y 427.758,Z 919.419,A -85,B 0,C 180,E1 21433.806,E2 21433.806} C_VEL
LIN {X 0,Y 432.786,Z 935.348,A -85,B 0,C 180,E1 21439.06,E2 21439.06} C_VEL
LIN {X 0,Y 438.014,Z 956.447,A -85,B 0,C 180,E1 21444.194,E2 21444.194} C_VEL
LIN {X 0,Y 438.376,Z 960.573,A -85,B 0,C 180,E1 21444.916,E2 21444.916} C_VEL
LIN {X 0,Y 419.707,Z 1004.527,A -85,B 0,C 180,E1 21447.777,E2 21447.777} C_VEL
LIN {X 0,Y 399.54,Z 1044.907,A -85,B 0,C 180,E1 21451.423,E2 21451.423} C_VEL
LIN {X 0,Y 377.966,Z 1082.376,A -85,B 0,C 180,E1 21456.129,E2 21456.129} C_VEL
LIN {X 0,Y 357.764,Z 1115.142,A -85,B 0,C 180,E1 21461.846,E2 21461.846} C_VEL
LIN {X 0,Y 339.069,Z 1144.226,A -85,B 0,C 180,E1 21468.977,E2 21468.977} C_VEL
LIN {X 0,Y 325.103,Z 1167.142,A -85,B 0,C 180,E1 21476.806,E2 21476.806} C_VEL
LIN {X 0,Y 315.654,Z 1184.766,A -85,B 0,C 180,E1 21485.469,E2 21485.469} C_VEL
LIN {X 0,Y 311.466,Z 1195.429,A -85,B 0,C 180,E1 21493.075,E2 21493.075} C_VEL
LIN {X 0,Y 310.078,Z 1200.903,A -85,B 0,C 180,E1 21498.758,E2 21498.758} C_VEL
LIN {X 0,Y 309.62,Z 1204.831,A -85,B 0,C 180,E1 21507.201,E2 21507.201} C_VEL
LIN {X 0,Y 309.703,Z 1204.835,A -85,B 0,C 180,E1 21512.795,E2 21512.795} C_VEL
LIN {X 0,Y 310.072,Z 1200.913,A -85,B 0,C 180,E1 21521.24,E2 21521.24} C_VEL
LIN {X 0,Y 312.718,Z 1191.964,A -85,B 0,C 180,E1 21529.769,E2 21529.769} C_VEL
LIN {X 0,Y 319.745,Z 1176.74,A -85,B 0,C 180,E1 21538.881,E2 21538.881} C_VEL
LIN {X 0,Y 331.064,Z 1157.2,A -85,B 0,C 180,E1 21546.928,E2 21546.928} C_VEL
LIN {X 0,Y 348.272,Z 1129.972,A -85,B 0,C 180,E1 21554.833,E2 21554.833} C_VEL
LIN {X 0,Y 367.059,Z 1100.395,A -85,B 0,C 180,E1 21560.97,E2 21560.97} C_VEL
LIN {X 0,Y 389.485,Z 1062.983,A -85,B 0,C 180,E1 21566.525,E2 21566.525} C_VEL
LIN {X 0,Y 410.401,Z 1023.985,A -85,B 0,C 180,E1 21570.631,E2 21570.631} C_VEL
LIN {X 0,Y 430.049,Z 981.675,A -85,B 0,C 180,E1 21573.828,E2 21573.828} C_VEL
LIN {X 0,Y 438.706,Z 959.68,A -85,B 0,C 180,E1 21575.17,E2 21575.17} C_VEL
LIN {X 0,Y 433.671,Z 938.332,A -85,B 0,C 180,E1 21580.184,E2 21580.184} C_VEL
LIN {X 0,Y 430.114,Z 926.675,A -85,B 0,C 180,E1 21583.678,E2 21583.678} C_VEL
LIN {X 0,Y 427.549,Z 924.23,A -85,B 0,C 180,E1 21585.366,E2 21585.366} C_VEL
LIN {X 0,Y 423.018,Z 922.365,A -85,B 0,C 180,E1 21588.276,E2 21588.276} C_VEL
LIN {X 0,Y 419.8,Z 913.169,A -85,B 0,C 180,E1 21593.789,E2 21593.789} C_VEL
LIN {X 0,Y 418.835,Z 907.876,A -85,B 0,C 180,E1 21599.988,E2 21599.988} C_VEL
LIN {X 0,Y 418.496,Z 909.593,A -85,B 0,C 180,E1 21603.092,E2 21603.092} C_VEL
LIN {X 0,Y 419.977,Z 916.865,A -85,B 0,C 180,E1 21609.305,E2 21609.305} C_VEL
LIN {X 0,Y 423.135,Z 928.568,A -85,B 0,C 180,E1 21615.017,E2 21615.017} C_VEL
LIN {X 0,Y 426.775,Z 944.185,A -85,B 0,C 180,E1 21620.18,E2 21620.18} C_VEL
LIN {X 0,Y 429.974,Z 964.445,A -85,B 0,C 180,E1 21625.205,E2 21625.205} C_VEL
LIN {X 0,Y 410.337,Z 1006.668,A -85,B 0,C 180,E1 21628.375,E2 21628.375} C_VEL
LIN {X 0,Y 388.546,Z 1046.424,A -85,B 0,C 180,E1 21632.528,E2 21632.528} C_VEL
LIN {X 0,Y 366.944,Z 1080.76,A -85,B 0,C 180,E1 21637.56,E2 21637.56} C_VEL
LIN {X 0,Y 346.305,Z 1111.22,A -85,B 0,C 180,E1 21643.774,E2 21643.774} C_VEL
LIN {X 0,Y 328.665,Z 1136.202,A -85,B 0,C 180,E1 21651.023,E2 21651.023} C_VEL
LIN {X 0,Y 315.376,Z 1156.058,A -85,B 0,C 180,E1 21659.16,E2 21659.16} C_VEL
LIN {X 0,Y 307.683,Z 1169.22,A -85,B 0,C 180,E1 21666.866,E2 21666.866} C_VEL
LIN {X 0,Y 303.228,Z 1178.933,A -85,B 0,C 180,E1 21675.573,E2 21675.573} C_VEL
LIN {X 0,Y 301.959,Z 1182.877,A -85,B 0,C 180,E1 21681.367,E2 21681.367} C_VEL
LIN {X 0,Y 301.836,Z 1185.108,A -85,B 0,C 180,E1 21690.001,E2 21690.001} C_VEL
LIN {X 0,Y 302.031,Z 1182.812,A -85,B 0,C 180,E1 21698.634,E2 21698.634} C_VEL
LIN {X 0,Y 304.366,Z 1176.066,A -85,B 0,C 180,E1 21707.332,E2 21707.332} C_VEL
LIN {X 0,Y 310.907,Z 1163.501,A -85,B 0,C 180,E1 21716.718,E2 21716.718} C_VEL
LIN {X 0,Y 322.893,Z 1144.525,A -85,B 0,C 180,E1 21725.804,E2 21725.804} C_VEL
LIN {X 0,Y 339.474,Z 1120.811,A -85,B 0,C 180,E1 21733.628,E2 21733.628} C_VEL
LIN {X 0,Y 360.267,Z 1090.656,A -85,B 0,C 180,E1 21740.551,E2 21740.551} C_VEL
LIN {X 0,Y 381.301,Z 1058.172,A -85,B 0,C 180,E1 21745.823,E2 21745.823} C_VEL
LIN {X 0,Y 403.458,Z 1019.753,A -85,B 0,C 180,E1 21750.297,E2 21750.297} C_VEL
LIN {X 0,Y 422.787,Z 980.858,A -85,B 0,C 180,E1 21753.549,E2 21753.549} C_VEL
LIN {X 0,Y 429.871,Z 963.876,A -85,B 0,C 180,E1 21754.788,E2 21754.788} C_VEL
LIN {X 0,Y 426.537,Z 943.897,A -85,B 0,C 180,E1 21759.808,E2 21759.808} C_VEL
LIN {X 0,Y 422.904,Z 928.389,A -85,B 0,C 180,E1 21764.948,E2 21764.948} C_VEL
LIN {X 0,Y 420.232,Z 918.224,A -85,B 0,C 180,E1 21769.656,E2 21769.656} C_VEL
LIN {X 0,Y 418.394,Z 911.372,A -85,B 0,C 180,E1 21774.832,E2 21774.832} C_VEL
LIN {X 0,Y 418.527,Z 908.122,A -85,B 0,C 180,E1 21777.943,E2 21777.943} C_VEL
LIN {X 0,Y 418.75,Z 908.587,A -85,B 0,C 180,E1 21782.08,E2 21782.08} C_VEL
LIN {X 0,Y 420.64,Z 915.8,A -85,B 0,C 180,E1 21788.273,E2 21788.273} C_VEL
LIN {X 0,Y 424.388,Z 926.585,A -85,B 0,C 180,E1 21793.693,E2 21793.693} C_VEL
LIN {X 0,Y 428.984,Z 942.148,A -85,B 0,C 180,E1 21798.852,E2 21798.852} C_VEL
LIN {X 0,Y 433.504,Z 962.755,A -85,B 0,C 180,E1 21803.933,E2 21803.933} C_VEL
LIN {X 0,Y 432.939,Z 965.448,A -85,B 0,C 180,E1 21804.24,E2 21804.24} C_VEL
LIN {X 0,Y 413.256,Z 1009.974,A -85,B 0,C 180,E1 21807.221,E2 21807.221} C_VEL
LIN {X 0,Y 392.861,Z 1048.947,A -85,B 0,C 180,E1 21810.879,E2 21810.879} C_VEL
LIN {X 0,Y 370.31,Z 1086.71,A -85,B 0,C 180,E1 21815.793,E2 21815.793} C_VEL
LIN {X 0,Y 349.4,Z 1119.082,A -85,B 0,C 180,E1 21821.75,E2 21821.75} C_VEL
LIN {X 0,Y 330.114,Z 1148.071,A -85,B 0,C 180,E1 21829.244,E2 21829.244} C_VEL
LIN {X 0,Y 315.803,Z 1170.647,A -85,B 0,C 180,E1 21837.661,E2 21837.661} C_VEL
LIN {X 0,Y 306.764,Z 1187.672,A -85,B 0,C 180,E1 21846.79,E2 21846.79} C_VEL
LIN {X 0,Y 302.799,Z 1198.147,A -85,B 0,C 180,E1 21855.549,E2 21855.549} C_VEL
LIN {X 0,Y 301.789,Z 1202.433,A -85,B 0,C 180,E1 21861.359,E2 21861.359} C_VEL
LIN {X 0,Y 301.912,Z 1204.926,A -85,B 0,C 180,E1 21869.999,E2 21869.999} C_VEL
LIN {X 0,Y 301.675,Z 1203.744,A -85,B 0,C 180,E1 21875.748,E2 21875.748} C_VEL
LIN {X 0,Y 302.577,Z 1198.977,A -85,B 0,C 180,E1 21883.501,E2 21883.501} C_VEL
LIN {X 0,Y 306.305,Z 1188.714,A -85,B 0,C 180,E1 21892.477,E2 21892.477} C_VEL
LIN {X 0,Y 314.319,Z 1173.246,A -85,B 0,C 180,E1 21901.187,E2 21901.187} C_VEL
LIN {X 0,Y 328.68,Z 1150.266,A -85,B 0,C 180,E1 21910.063,E2 21910.063} C_VEL
LIN {X 0,Y 346.654,Z 1123.206,A -85,B 0,C 180,E1 21917.356,E2 21917.356} C_VEL
LIN {X 0,Y 368.576,Z 1089.746,A -85,B 0,C 180,E1 21923.748,E2 21923.748} C_VEL
LIN {X 0,Y 390.375,Z 1053.349,A -85,B 0,C 180,E1 21928.65,E2 21928.65} C_VEL
LIN {X 0,Y 411.538,Z 1013.746,A -85,B 0,C 180,E1 21932.503,E2 21932.503} C_VEL
LIN {X 0,Y 431.577,Z 969.139,A -85,B 0,C 180,E1 21935.552,E2 21935.552} C_VEL
LIN {X 0,Y 433.683,Z 963.551,A -85,B 0,C 180,E1 21935.924,E2 21935.924} C_VEL
LIN {X 0,Y 429.047,Z 942.363,A -85,B 0,C 180,E1 21941.151,E2 21941.151} C_VEL
LIN {X 0,Y 424.496,Z 927.064,A -85,B 0,C 180,E1 21946.247,E2 21946.247} C_VEL
LIN {X 0,Y 423.018,Z 922.365,A -85,B 0,C 180,E1 21948.276,E2 21948.276} C_VEL
LIN {X 0,Y 420.854,Z 921.263,A -85,B 0,C 180,E1 21950.027,E2 21950.027} C_VEL
LIN {X 0,Y 417.172,Z 921.517,A -85,B 0,C 180,E1 21953.008,E2 21953.008} C_VEL
LIN {X 0,Y 415.965,Z 915.248,A -85,B 0,C 180,E1 21959.988,E2 21959.988} C_VEL
LIN {X 0,Y 415.608,Z 917.022,A -85,B 0,C 180,E1 21963.114,E2 21963.114} C_VEL
LIN {X 0,Y 416.729,Z 924.305,A -85,B 0,C 180,E1 21969.378,E2 21969.378} C_VEL
LIN {X 0,Y 419.674,Z 936.294,A -85,B 0,C 180,E1 21975.144,E2 21975.144} C_VEL
LIN {X 0,Y 422.934,Z 952.496,A -85,B 0,C 180,E1 21980.442,E2 21980.442} C_VEL
LIN {X 0,Y 425.024,Z 968.349,A -85,B 0,C 180,E1 21984.447,E2 21984.447} C_VEL
LIN {X 0,Y 403.826,Z 1012.18,A -85,B 0,C 180,E1 21987.847,E2 21987.847} C_VEL
LIN {X 0,Y 382.795,Z 1048.992,A -85,B 0,C 180,E1 21991.793,E2 21991.793} C_VEL
LIN {X 0,Y 359.902,Z 1084.17,A -85,B 0,C 180,E1 21997.086,E2 21997.086} C_VEL
LIN {X 0,Y 339.163,Z 1113.481,A -85,B 0,C 180,E1 22003.279,E2 22003.279} C_VEL
LIN {X 0,Y 319.788,Z 1139.972,A -85,B 0,C 180,E1 22011.338,E2 22011.338} C_VEL
LIN {X 0,Y 306.689,Z 1158.844,A -85,B 0,C 180,E1 22019.71,E2 22019.71} C_VEL
LIN {X 0,Y 298.227,Z 1173.209,A -85,B 0,C 180,E1 22029.227,E2 22029.227} C_VEL
LIN {X 0,Y 294.662,Z 1181.491,A -85,B 0,C 180,E1 22038.164,E2 22038.164} C_VEL
LIN {X 0,Y 293.745,Z 1185.058,A -85,B 0,C 180,E1 22047.053,E2 22047.053} C_VEL
LIN {X 0,Y 293.838,Z 1185.043,A -85,B 0,C 180,E1 22052.949,E2 22052.949} C_VEL
LIN {X 0,Y 294.72,Z 1181.423,A -85,B 0,C 180,E1 22061.836,E2 22061.836} C_VEL
LIN {X 0,Y 298.269,Z 1173.077,A -85,B 0,C 180,E1 22070.773,E2 22070.773} C_VEL
LIN {X 0,Y 306.829,Z 1158.597,A -85,B 0,C 180,E1 22080.317,E2 22080.317} C_VEL
LIN {X 0,Y 320.071,Z 1139.556,A -85,B 0,C 180,E1 22088.698,E2 22088.698} C_VEL
LIN {X 0,Y 339.516,Z 1112.982,A -85,B 0,C 180,E1 22096.735,E2 22096.735} C_VEL
LIN {X 0,Y 360.072,Z 1083.766,A -85,B 0,C 180,E1 22102.882,E2 22102.882} C_VEL
LIN {X 0,Y 382.673,Z 1049.072,A -85,B 0,C 180,E1 22108.083,E2 22108.083} C_VEL
LIN {X 0,Y 403.406,Z 1012.838,A -85,B 0,C 180,E1 22111.977,E2 22111.977} C_VEL
LIN {X 0,Y 424.401,Z 969.684,A -85,B 0,C 180,E1 22115.324,E2 22115.324} C_VEL
LIN {X 0,Y 424.396,Z 963.705,A -85,B 0,C 180,E1 22116.528,E2 22116.528} C_VEL
LIN {X 0,Y 421.353,Z 944.843,A -85,B 0,C 180,E1 22121.726,E2 22121.726} C_VEL
LIN {X 0,Y 417.996,Z 929.779,A -85,B 0,C 180,E1 22127.486,E2 22127.486} C_VEL
LIN {X 0,Y 415.948,Z 920.832,A -85,B 0,C 180,E1 22132.711,E2 22132.711} C_VEL
LIN {X 0,Y 415.631,Z 915.567,A -85,B 0,C 180,E1 22137.929,E2 22137.929} C_VEL
LIN {X 0,Y 415.843,Z 916.06,A -85,B 0,C 180,E1 22142.094,E2 22142.094} C_VEL
LIN {X 0,Y 417.586,Z 923.316,A -85,B 0,C 180,E1 22148.334,E2 22148.334} C_VEL
LIN {X 0,Y 421.071,Z 934.306,A -85,B 0,C 180,E1 22153.803,E2 22153.803} C_VEL
LIN {X 0,Y 424.931,Z 948.929,A -85,B 0,C 180,E1 22158.676,E2 22158.676} C_VEL
LIN {X 0,Y 428.59,Z 967.054,A -85,B 0,C 180,E1 22163.272,E2 22163.272} C_VEL
LIN {X 0,Y 408.149,Z 1012.719,A -85,B 0,C 180,E1 22166.442,E2 22166.442} C_VEL
LIN {X 0,Y 386.821,Z 1051.858,A -85,B 0,C 180,E1 22170.194,E2 22170.194} C_VEL
LIN {X 0,Y 364.2,Z 1088.591,A -85,B 0,C 180,E1 22175.07,E2 22175.07} C_VEL
LIN {X 0,Y 342.027,Z 1121.502,A -85,B 0,C 180,E1 22181.314,E2 22181.314} C_VEL
LIN {X 0,Y 323.436,Z 1148.47,A -85,B 0,C 180,E1 22188.492,E2 22188.492} C_VEL
LIN {X 0,Y 308.135,Z 1171.499,A -85,B 0,C 180,E1 22197.352,E2 22197.352} C_VEL
LIN {X 0,Y 299.231,Z 1187.402,A -85,B 0,C 180,E1 22206.17,E2 22206.17} C_VEL
LIN {X 0,Y 295.012,Z 1197.883,A -85,B 0,C 180,E1 22215.159,E2 22215.159} C_VEL
LIN {X 0,Y 293.897,Z 1202.17,A -85,B 0,C 180,E1 22221.125,E2 22221.125} C_VEL
LIN {X 0,Y 294.011,Z 1204.666,A -85,B 0,C 180,E1 22229.999,E2 22229.999} C_VEL
LIN {X 0,Y 293.764,Z 1203.483,A -85,B 0,C 180,E1 22235.904,E2 22235.904} C_VEL
LIN {X 0,Y 294.503,Z 1199.592,A -85,B 0,C 180,E1 22242.819,E2 22242.819} C_VEL
LIN {X 0,Y 297.408,Z 1191.43,A -85,B 0,C 180,E1 22250.833,E2 22250.833} C_VEL
LIN {X 0,Y 305.108,Z 1176.589,A -85,B 0,C 180,E1 22260.175,E2 22260.175} C_VEL
LIN {X 0,Y 318.268,Z 1155.964,A -85,B 0,C 180,E1 22268.982,E2 22268.982} C_VEL
LIN {X 0,Y 337.046,Z 1128.773,A -85,B 0,C 180,E1 22277.013,E2 22277.013} C_VEL
LIN {X 0,Y 357.895,Z 1098.166,A -85,B 0,C 180,E1 22283.341,E2 22283.341} C_VEL
LIN {X 0,Y 380.643,Z 1062.435,A -85,B 0,C 180,E1 22288.599,E2 22288.599} C_VEL
LIN {X 0,Y 402.822,Z 1023.076,A -85,B 0,C 180,E1 22292.694,E2 22292.694} C_VEL
LIN {X 0,Y 424.263,Z 978.681,A -85,B 0,C 180,E1 22295.961,E2 22295.961} C_VEL
LIN {X 0,Y 428.615,Z 967.31,A -85,B 0,C 180,E1 22296.724,E2 22296.724} C_VEL
LIN {X 0,Y 424.593,Z 947.345,A -85,B 0,C 180,E1 22301.846,E2 22301.846} C_VEL
LIN {X 0,Y 420.186,Z 931.383,A -85,B 0,C 180,E1 22307.528,E2 22307.528} C_VEL
LIN {X 0,Y 417.172,Z 921.517,A -85,B 0,C 180,E1 22313.008,E2 22313.008} C_VEL
LIN {X 0,Y 416.163,Z 921.321,A -85,B 0,C 180,E1 22314.202,E2 22314.202} C_VEL
LIN {X 0,Y 412.85,Z 924.118,A -85,B 0,C 180,E1 22317.499,E2 22317.499} C_VEL
LIN {X 0,Y 412.832,Z 923.886,A -85,B 0,C 180,E1 22317.802,E2 22317.802} C_VEL
LIN {X 0,Y 412.895,Z 922.553,A -85,B 0,C 180,E1 22319.988,E2 22319.988} C_VEL
LIN {X 0,Y 412.401,Z 924.345,A -85,B 0,C 180,E1 22323.138,E2 22323.138} C_VEL
LIN {X 0,Y 413.418,Z 931.502,A -85,B 0,C 180,E1 22329.293,E2 22329.293} C_VEL
LIN {X 0,Y 416.019,Z 943.813,A -85,B 0,C 180,E1 22335.254,E2 22335.254} C_VEL
LIN {X 0,Y 418.544,Z 958.764,A -85,B 0,C 180,E1 22340.168,E2 22340.168} C_VEL
LIN {X 0,Y 420.031,Z 972.463,A -85,B 0,C 180,E1 22343.73,E2 22343.73} C_VEL
LIN {X 0,Y 398.602,Z 1015.31,A -85,B 0,C 180,E1 22347.084,E2 22347.084} C_VEL
LIN {X 0,Y 376.53,Z 1052.361,A -85,B 0,C 180,E1 22351.146,E2 22351.146} C_VEL
LIN {X 0,Y 352.69,Z 1087.828,A -85,B 0,C 180,E1 22356.632,E2 22356.632} C_VEL
LIN {X 0,Y 330.719,Z 1117.474,A -85,B 0,C 180,E1 22363.238,E2 22363.238} C_VEL
LIN {X 0,Y 312.201,Z 1141.906,A -85,B 0,C 180,E1 22371.009,E2 22371.009} C_VEL
LIN {X 0,Y 298.773,Z 1160.34,A -85,B 0,C 180,E1 22379.619,E2 22379.619} C_VEL
LIN {X 0,Y 290.126,Z 1174.578,A -85,B 0,C 180,E1 22389.57,E2 22389.57} C_VEL
LIN {X 0,Y 286.835,Z 1181.754,A -85,B 0,C 180,E1 22397.836,E2 22397.836} C_VEL
LIN {X 0,Y 285.859,Z 1185.318,A -85,B 0,C 180,E1 22406.971,E2 22406.971} C_VEL
LIN {X 0,Y 285.937,Z 1185.303,A -85,B 0,C 180,E1 22413.031,E2 22413.031} C_VEL
LIN {X 0,Y 286.894,Z 1181.686,A -85,B 0,C 180,E1 22422.164,E2 22422.164} C_VEL
LIN {X 0,Y 290.696,Z 1173.344,A -85,B 0,C 180,E1 22431.34,E2 22431.34} C_VEL
LIN {X 0,Y 299.67,Z 1158.998,A -85,B 0,C 180,E1 22441.037,E2 22441.037} C_VEL
LIN {X 0,Y 313.688,Z 1139.883,A -85,B 0,C 180,E1 22449.612,E2 22449.612} C_VEL
LIN {X 0,Y 334.016,Z 1113.12,A -85,B 0,C 180,E1 22457.803,E2 22457.803} C_VEL
LIN {X 0,Y 356.126,Z 1082.682,A -85,B 0,C 180,E1 22464.174,E2 22464.174} C_VEL
LIN {X 0,Y 378.611,Z 1049.069,A -85,B 0,C 180,E1 22469.165,E2 22469.165} C_VEL
LIN {X 0,Y 399.943,Z 1012.556,A -85,B 0,C 180,E1 22473.056,E2 22473.056} C_VEL
LIN {X 0,Y 419.921,Z 972.188,A -85,B 0,C 180,E1 22476.218,E2 22476.218} C_VEL
LIN {X 0,Y 417.74,Z 954.488,A -85,B 0,C 180,E1 22481.016,E2 22481.016} C_VEL
LIN {X 0,Y 415.028,Z 939.64,A -85,B 0,C 180,E1 22486.324,E2 22486.324} C_VEL
LIN {X 0,Y 412.978,Z 929.716,A -85,B 0,C 180,E1 22491.597,E2 22491.597} C_VEL
LIN {X 0,Y 412.496,Z 922.927,A -85,B 0,C 180,E1 22497.913,E2 22497.913} C_VEL
LIN {X 0,Y 412.679,Z 922.406,A -85,B 0,C 180,E1 22500.012,E2 22500.012} C_VEL
LIN {X 0,Y 413.08,Z 926.701,A -85,B 0,C 180,E1 22505.259,E2 22505.259} C_VEL
LIN {X 0,Y 415.494,Z 934.282,A -85,B 0,C 180,E1 22510.488,E2 22510.488} C_VEL
LIN {X 0,Y 418.887,Z 946.784,A -85,B 0,C 180,E1 22515.708,E2 22515.708} C_VEL
LIN {X 0,Y 422.602,Z 964.8,A -85,B 0,C 180,E1 22520.961,E2 22520.961} C_VEL
LIN {X 0,Y 423.362,Z 972.411,A -85,B 0,C 180,E1 22522.678,E2 22522.678} C_VEL
LIN {X 0,Y 403.206,Z 1015.003,A -85,B 0,C 180,E1 22525.617,E2 22525.617} C_VEL
LIN {X 0,Y 380.405,Z 1055.52,A -85,B 0,C 180,E1 22529.576,E2 22529.576} C_VEL
LIN {X 0,Y 358.291,Z 1090.088,A -85,B 0,C 180,E1 22534.274,E2 22534.274} C_VEL
LIN {X 0,Y 334.822,Z 1123.716,A -85,B 0,C 180,E1 22540.813,E2 22540.813} C_VEL
LIN {X 0,Y 316.118,Z 1149.669,A -85,B 0,C 180,E1 22547.991,E2 22547.991} C_VEL
LIN {X 0,Y 300.18,Z 1172.796,A -85,B 0,C 180,E1 22557.236,E2 22557.236} C_VEL
LIN {X 0,Y 291.195,Z 1188.152,A -85,B 0,C 180,E1 22566.284,E2 22566.284} C_VEL
LIN {X 0,Y 287.203,Z 1197.617,A -85,B 0,C 180,E1 22574.746,E2 22574.746} C_VEL
LIN {X 0,Y 286.032,Z 1201.909,A -85,B 0,C 180,E1 22580.879,E2 22580.879} C_VEL
LIN {X 0,Y 286.125,Z 1204.407,A -85,B 0,C 180,E1 22589.998,E2 22589.998} C_VEL
LIN {X 0,Y 285.856,Z 1203.222,A -85,B 0,C 180,E1 22596.067,E2 22596.067} C_VEL
LIN {X 0,Y 286.661,Z 1199.328,A -85,B 0,C 180,E1 22603.176,E2 22603.176} C_VEL
LIN {X 0,Y 289.79,Z 1191.163,A -85,B 0,C 180,E1 22611.407,E2 22611.407} C_VEL
LIN {X 0,Y 298.325,Z 1175.765,A -85,B 0,C 180,E1 22621.277,E2 22621.277} C_VEL
LIN {X 0,Y 311.791,Z 1155.691,A -85,B 0,C 180,E1 22629.952,E2 22629.952} C_VEL
LIN {X 0,Y 331.909,Z 1127.836,A -85,B 0,C 180,E1 22638.239,E2 22638.239} C_VEL
LIN {X 0,Y 353.761,Z 1096.779,A -85,B 0,C 180,E1 22644.612,E2 22644.612} C_VEL
LIN {X 0,Y 377.61,Z 1060.355,A -85,B 0,C 180,E1 22649.889,E2 22649.889} C_VEL
LIN {X 0,Y 401.146,Z 1018.989,A -85,B 0,C 180,E1 22654.073,E2 22654.073} C_VEL
LIN {X 0,Y 421.6,Z 977.045,A -85,B 0,C 180,E1 22657.053,E2 22657.053} C_VEL
LIN {X 0,Y 423.467,Z 972.59,A -85,B 0,C 180,E1 22657.31,E2 22657.31} C_VEL
LIN {X 0,Y 421.228,Z 957.141,A -85,B 0,C 180,E1 22661.154,E2 22661.154} C_VEL
LIN {X 0,Y 417.776,Z 942.43,A -85,B 0,C 180,E1 22666.021,E2 22666.021} C_VEL
LIN {X 0,Y 414.47,Z 930.968,A -85,B 0,C 180,E1 22671.603,E2 22671.603} C_VEL
LIN {X 0,Y 412.832,Z 923.886,A -85,B 0,C 180,E1 22677.802,E2 22677.802} C_VEL
LIN {X 0,Y 411.872,Z 924.977,A -85,B 0,C 180,E1 22679.604,E2 22679.604} C_VEL
LIN {X 0,Y 409.29,Z 931.058,A -85,B 0,C 180,E1 22682.595,E2 22682.595} C_VEL
LIN {X 0,Y 409.779,Z 937.449,A -85,B 0,C 180,E1 22688.469,E2 22688.469} C_VEL
LIN {X 0,Y 411.807,Z 948.8,A -85,B 0,C 180,E1 22694.326,E2 22694.326} C_VEL
LIN {X 0,Y 413.993,Z 963.586,A -85,B 0,C 180,E1 22699.471,E2 22699.471} C_VEL
LIN {X 0,Y 415.104,Z 976.558,A -85,B 0,C 180,E1 22702.99,E2 22702.99} C_VEL
LIN {X 0,Y 394.103,Z 1017.202,A -85,B 0,C 180,E1 22706.185,E2 22706.185} C_VEL
LIN {X 0,Y 370.351,Z 1055.669,A -85,B 0,C 180,E1 22710.467,E2 22710.467} C_VEL
LIN {X 0,Y 347.085,Z 1089.174,A -85,B 0,C 180,E1 22715.751,E2 22715.751} C_VEL
LIN {X 0,Y 324.49,Z 1118.564,A -85,B 0,C 180,E1 22722.402,E2 22722.402} C_VEL
LIN {X 0,Y 305.865,Z 1142.174,A -85,B 0,C 180,E1 22730.041,E2 22730.041} C_VEL
LIN {X 0,Y 291.741,Z 1160.608,A -85,B 0,C 180,E1 22738.806,E2 22738.806} C_VEL
LIN {X 0,Y 283.114,Z 1173.74,A -85,B 0,C 180,E1 22748.062,E2 22748.062} C_VEL
LIN {X 0,Y 279.006,Z 1182.016,A -85,B 0,C 180,E1 22757.49,E2 22757.49} C_VEL
LIN {X 0,Y 277.955,Z 1185.577,A -85,B 0,C 180,E1 22766.885,E2 22766.885} C_VEL
LIN {X 0,Y 278.031,Z 1185.563,A -85,B 0,C 180,E1 22773.117,E2 22773.117} C_VEL
LIN {X 0,Y 279.065,Z 1181.949,A -85,B 0,C 180,E1 22782.511,E2 22782.511} C_VEL
LIN {X 0,Y 283.15,Z 1173.611,A -85,B 0,C 180,E1 22791.938,E2 22791.938} C_VEL
LIN {X 0,Y 292.666,Z 1159.269,A -85,B 0,C 180,E1 22801.865,E2 22801.865} C_VEL
LIN {X 0,Y 307.421,Z 1140.154,A -85,B 0,C 180,E1 22810.585,E2 22810.585} C_VEL
LIN {X 0,Y 327.603,Z 1114.568,A -85,B 0,C 180,E1 22818.554,E2 22818.554} C_VEL
LIN {X 0,Y 349.325,Z 1085.854,A -85,B 0,C 180,E1 22824.747,E2 22824.747} C_VEL
LIN {X 0,Y 373.449,Z 1050.922,A -85,B 0,C 180,E1 22830.029,E2 22830.029} C_VEL
LIN {X 0,Y 395.113,Z 1015.135,A -85,B 0,C 180,E1 22833.886,E2 22833.886} C_VEL
LIN {X 0,Y 414.959,Z 976.297,A -85,B 0,C 180,E1 22836.966,E2 22836.966} C_VEL
LIN {X 0,Y 413.147,Z 958.58,A -85,B 0,C 180,E1 22841.986,E2 22841.986} C_VEL
LIN {X 0,Y 410.917,Z 944.817,A -85,B 0,C 180,E1 22847.267,E2 22847.267} C_VEL
LIN {X 0,Y 409.425,Z 935.504,A -85,B 0,C 180,E1 22852.672,E2 22852.672} C_VEL
LIN {X 0,Y 409.262,Z 930.245,A -85,B 0,C 180,E1 22857.897,E2 22857.897} C_VEL
LIN {X 0,Y 409.487,Z 929.621,A -85,B 0,C 180,E1 22860.012,E2 22860.012} C_VEL
LIN {X 0,Y 410.274,Z 935.071,A -85,B 0,C 180,E1 22866.355,E2 22866.355} C_VEL
LIN {X 0,Y 412.831,Z 944.666,A -85,B 0,C 180,E1 22871.983,E2 22871.983} C_VEL
LIN {X 0,Y 416.16,Z 959.091,A -85,B 0,C 180,E1 22877.321,E2 22877.321} C_VEL
LIN {X 0,Y 418.657,Z 974.989,A -85,B 0,C 180,E1 22881.681,E2 22881.681} C_VEL
LIN {X 0,Y 415.355,Z 983.224,A -85,B 0,C 180,E1 22882.33,E2 22882.33} C_VEL
LIN {X 0,Y 392.833,Z 1027.41,A -85,B 0,C 180,E1 22885.632,E2 22885.632} C_VEL
LIN {X 0,Y 369.504,Z 1066.093,A -85,B 0,C 180,E1 22889.791,E2 22889.791} C_VEL
LIN {X 0,Y 346.034,Z 1100.747,A -85,B 0,C 180,E1 22895.033,E2 22895.033} C_VEL
LIN {X 0,Y 323.551,Z 1131.248,A -85,B 0,C 180,E1 22901.644,E2 22901.644} C_VEL
LIN {X 0,Y 304.016,Z 1157.346,A -85,B 0,C 180,E1 22909.745,E2 22909.745} C_VEL
LIN {X 0,Y 289.57,Z 1178.016,A -85,B 0,C 180,E1 22919.296,E2 22919.296} C_VEL
LIN {X 0,Y 281.687,Z 1191.998,A -85,B 0,C 180,E1 22928.88,E2 22928.88} C_VEL
LIN {X 0,Y 278.651,Z 1199.87,A -85,B 0,C 180,E1 22937.507,E2 22937.507} C_VEL
LIN {X 0,Y 277.995,Z 1203.791,A -85,B 0,C 180,E1 22946.882,E2 22946.882} C_VEL
LIN {X 0,Y 278.094,Z 1203.797,A -85,B 0,C 180,E1 22953.113,E2 22953.113} C_VEL
LIN {X 0,Y 278.649,Z 1199.86,A -85,B 0,C 180,E1 22962.527,E2 22962.527} C_VEL
LIN {X 0,Y 282.184,Z 1190.895,A -85,B 0,C 180,E1 22972.014,E2 22972.014} C_VEL
LIN {X 0,Y 291.265,Z 1175.494,A -85,B 0,C 180,E1 22982.124,E2 22982.124} C_VEL
LIN {X 0,Y 305.417,Z 1155.46,A -85,B 0,C 180,E1 22990.942,E2 22990.942} C_VEL
LIN {X 0,Y 325.699,Z 1128.475,A -85,B 0,C 180,E1 22999.098,E2 22999.098} C_VEL
LIN {X 0,Y 348.244,Z 1097.627,A -85,B 0,C 180,E1 23005.531,E2 23005.531} C_VEL
LIN {X 0,Y 373.217,Z 1060.593,A -85,B 0,C 180,E1 23010.919,E2 23010.919} C_VEL
LIN {X 0,Y 396.254,Z 1021.272,A -85,B 0,C 180,E1 23014.916,E2 23014.916} C_VEL
LIN {X 0,Y 418.233,Z 977.437,A -85,B 0,C 180,E1 23018.036,E2 23018.036} C_VEL
LIN {X 0,Y 418.727,Z 975.155,A -85,B 0,C 180,E1 23018.322,E2 23018.322} C_VEL
LIN {X 0,Y 415.573,Z 956.406,A -85,B 0,C 180,E1 23023.622,E2 23023.622} C_VEL
LIN {X 0,Y 412.619,Z 943.713,A -85,B 0,C 180,E1 23028.586,E2 23028.586} C_VEL
LIN {X 0,Y 410.369,Z 935.043,A -85,B 0,C 180,E1 23033.831,E2 23033.831} C_VEL
LIN {X 0,Y 409.693,Z 929.792,A -85,B 0,C 180,E1 23039.988,E2 23039.988} C_VEL
LIN {X 0,Y 409.29,Z 931.058,A -85,B 0,C 180,E1 23042.595,E2 23042.595} C_VEL
LIN {X 0,Y 407.493,Z 936.88,A -85,B 0,C 180,E1 23044.904,E2 23044.904} C_VEL
LIN {X 0,Y 405.989,Z 942.864,A -85,B 0,C 180,E1 23047.226,E2 23047.226} C_VEL
LIN {X 0,Y 407.607,Z 953.782,A -85,B 0,C 180,E1 23053.383,E2 23053.383} C_VEL
LIN {X 0,Y 409.318,Z 967.073,A -85,B 0,C 180,E1 23058.332,E2 23058.332} C_VEL
LIN {X 0,Y 410.195,Z 980.143,A -85,B 0,C 180,E1 23062.091,E2 23062.091} C_VEL
LIN {X 0,Y 388.779,Z 1020.498,A -85,B 0,C 180,E1 23065.413,E2 23065.413} C_VEL
LIN {X 0,Y 363.631,Z 1059.895,A -85,B 0,C 180,E1 23069.892,E2 23069.892} C_VEL
LIN {X 0,Y 340.415,Z 1091.883,A -85,B 0,C 180,E1 23075.114,E2 23075.114} C_VEL
LIN {X 0,Y 316.516,Z 1121.92,A -85,B 0,C 180,E1 23082.151,E2 23082.151} C_VEL
LIN {X 0,Y 297.861,Z 1144.456,A -85,B 0,C 180,E1 23089.877,E2 23089.877} C_VEL
LIN {X 0,Y 282.699,Z 1163.627,A -85,B 0,C 180,E1 23099.593,E2 23099.593} C_VEL
LIN {X 0,Y 274.414,Z 1176.008,A -85,B 0,C 180,E1 23109.341,E2 23109.341} C_VEL
LIN {X 0,Y 271.208,Z 1182.278,A -85,B 0,C 180,E1 23117.124,E2 23117.124} C_VEL
LIN {X 0,Y 270.067,Z 1185.836,A -85,B 0,C 180,E1 23126.794,E2 23126.794} C_VEL
LIN {X 0,Y 270.134,Z 1185.823,A -85,B 0,C 180,E1 23133.208,E2 23133.208} C_VEL
LIN {X 0,Y 271.267,Z 1182.212,A -85,B 0,C 180,E1 23142.876,E2 23142.876} C_VEL
LIN {X 0,Y 275.641,Z 1173.878,A -85,B 0,C 180,E1 23152.568,E2 23152.568} C_VEL
LIN {X 0,Y 285.848,Z 1159.405,A -85,B 0,C 180,E1 23162.812,E2 23162.812} C_VEL
LIN {X 0,Y 301.299,Z 1140.311,A -85,B 0,C 180,E1 23171.648,E2 23171.648} C_VEL
LIN {X 0,Y 323.248,Z 1113.662,A -85,B 0,C 180,E1 23179.953,E2 23179.953} C_VEL
LIN {X 0,Y 346.587,Z 1083.538,A -85,B 0,C 180,E1 23186.308,E2 23186.308} C_VEL
LIN {X 0,Y 371.679,Z 1047.888,A -85,B 0,C 180,E1 23191.548,E2 23191.548} C_VEL
LIN {X 0,Y 394.536,Z 1010.152,A -85,B 0,C 180,E1 23195.41,E2 23195.41} C_VEL
LIN {X 0,Y 409.688,Z 981.461,A -85,B 0,C 180,E1 23197.617,E2 23197.617} C_VEL
LIN {X 0,Y 409.259,Z 968.25,A -85,B 0,C 180,E1 23201.209,E2 23201.209} C_VEL
LIN {X 0,Y 407.427,Z 953.478,A -85,B 0,C 180,E1 23206.611,E2 23206.611} C_VEL
LIN {X 0,Y 405.855,Z 942.673,A -85,B 0,C 180,E1 23212.657,E2 23212.657} C_VEL
LIN {X 0,Y 405.976,Z 937.537,A -85,B 0,C 180,E1 23217.88,E2 23217.88} C_VEL
LIN {X 0,Y 406.284,Z 936.847,A -85,B 0,C 180,E1 23220.012,E2 23220.012} C_VEL
LIN {X 0,Y 406.857,Z 942.348,A -85,B 0,C 180,E1 23226.409,E2 23226.409} C_VEL
LIN {X 0,Y 409.294,Z 952.52,A -85,B 0,C 180,E1 23232.268,E2 23232.268} C_VEL
LIN {X 0,Y 411.848,Z 965.499,A -85,B 0,C 180,E1 23237.08,E2 23237.08} C_VEL
LIN {X 0,Y 413.763,Z 979.304,A -85,B 0,C 180,E1 23240.947,E2 23240.947} C_VEL
LIN {X 0,Y 394.061,Z 1018.67,A -85,B 0,C 180,E1 23243.836,E2 23243.836} C_VEL
LIN {X 0,Y 370.192,Z 1058.796,A -85,B 0,C 180,E1 23247.809,E2 23247.809} C_VEL
LIN {X 0,Y 347.142,Z 1092.363,A -85,B 0,C 180,E1 23252.497,E2 23252.497} C_VEL
LIN {X 0,Y 322.687,Z 1125.168,A -85,B 0,C 180,E1 23259.049,E2 23259.049} C_VEL
LIN {X 0,Y 302.208,Z 1151.289,A -85,B 0,C 180,E1 23266.652,E2 23266.652} C_VEL
LIN {X 0,Y 285.323,Z 1173.802,A -85,B 0,C 180,E1 23276.212,E2 23276.212} C_VEL
LIN {X 0,Y 275.667,Z 1188.609,A -85,B 0,C 180,E1 23285.723,E2 23285.723} C_VEL
LIN {X 0,Y 271.173,Z 1198.344,A -85,B 0,C 180,E1 23295.476,E2 23295.476} C_VEL
LIN {X 0,Y 270.027,Z 1202.693,A -85,B 0,C 180,E1 23303.572,E2 23303.572} C_VEL
LIN {X 0,Y 270.339,Z 1203.889,A -85,B 0,C 180,E1 23309.998,E2 23309.998} C_VEL
LIN {X 0,Y 270.039,Z 1202.7,A -85,B 0,C 180,E1 23316.424,E2 23316.424} C_VEL
LIN {X 0,Y 271.167,Z 1198.361,A -85,B 0,C 180,E1 23324.521,E2 23324.521} C_VEL
LIN {X 0,Y 275.682,Z 1188.636,A -85,B 0,C 180,E1 23334.272,E2 23334.272} C_VEL
LIN {X 0,Y 285.303,Z 1173.846,A -85,B 0,C 180,E1 23343.787,E2 23343.787} C_VEL
LIN {X 0,Y 302.229,Z 1151.333,A -85,B 0,C 180,E1 23353.348,E2 23353.348} C_VEL
LIN {X 0,Y 322.686,Z 1125.272,A -85,B 0,C 180,E1 23360.945,E2 23360.945} C_VEL
LIN {X 0,Y 347.167,Z 1092.495,A -85,B 0,C 180,E1 23367.491,E2 23367.491} C_VEL
LIN {X 0,Y 370.973,Z 1057.667,A -85,B 0,C 180,E1 23372.344,E2 23372.344} C_VEL
LIN {X 0,Y 395.736,Z 1015.917,A -85,B 0,C 180,E1 23376.408,E2 23376.408} C_VEL
LIN {X 0,Y 413.877,Z 979.956,A -85,B 0,C 180,E1 23378.93,E2 23378.93} C_VEL
LIN {X 0,Y 411.334,Z 962.52,A -85,B 0,C 180,E1 23383.996,E2 23383.996} C_VEL
LIN {X 0,Y 408.588,Z 949.412,A -85,B 0,C 180,E1 23389.332,E2 23389.332} C_VEL
LIN {X 0,Y 406.671,Z 941.413,A -85,B 0,C 180,E1 23394.657,E2 23394.657} C_VEL
LIN {X 0,Y 406.482,Z 937.021,A -85,B 0,C 180,E1 23399.988,E2 23399.988} C_VEL
LIN {X 0,Y 405.752,Z 940.814,A -85,B 0,C 180,E1 23405.329,E2 23405.329} C_VEL
LIN {X 0,Y 405.989,Z 942.864,A -85,B 0,C 180,E1 23407.226,E2 23407.226} C_VEL
LIN {X 0,Y 405.196,Z 947.555,A -85,B 0,C 180,E1 23408.953,E2 23408.953} C_VEL
LIN {X 0,Y 403.183,Z 957.423,A -85,B 0,C 180,E1 23411.75,E2 23411.75} C_VEL
LIN {X 0,Y 404.58,Z 969.265,A -85,B 0,C 180,E1 23416.691,E2 23416.691} C_VEL
LIN {X 0,Y 405.333,Z 984.13,A -85,B 0,C 180,E1 23421.251,E2 23421.251} C_VEL
LIN {X 0,Y 401.91,Z 991.306,A -85,B 0,C 180,E1 23421.904,E2 23421.904} C_VEL
LIN {X 0,Y 378.554,Z 1031.93,A -85,B 0,C 180,E1 23425.43,E2 23425.43} C_VEL
LIN {X 0,Y 354.702,Z 1067.076,A -85,B 0,C 180,E1 23429.758,E2 23429.758} C_VEL
LIN {X 0,Y 329.576,Z 1099.917,A -85,B 0,C 180,E1 23435.529,E2 23435.529} C_VEL
LIN {X 0,Y 307.053,Z 1126.821,A -85,B 0,C 180,E1 23442.424,E2 23442.424} C_VEL
LIN {X 0,Y 286.626,Z 1150.697,A -85,B 0,C 180,E1 23451.455,E2 23451.455} C_VEL
LIN {X 0,Y 272.278,Z 1168.219,A -85,B 0,C 180,E1 23461.757,E2 23461.757} C_VEL
LIN {X 0,Y 265.206,Z 1179.002,A -85,B 0,C 180,E1 23471.738,E2 23471.738} C_VEL
LIN {X 0,Y 262.622,Z 1184.183,A -85,B 0,C 180,E1 23480.062,E2 23480.062} C_VEL
LIN {X 0,Y 262.349,Z 1186.404,A -85,B 0,C 180,E1 23490.002,E2 23490.002} C_VEL
LIN {X 0,Y 262.687,Z 1184.123,A -85,B 0,C 180,E1 23499.939,E2 23499.939} C_VEL
LIN {X 0,Y 266.072,Z 1177.395,A -85,B 0,C 180,E1 23509.925,E2 23509.925} C_VEL
LIN {X 0,Y 274.836,Z 1164.992,A -85,B 0,C 180,E1 23520.462,E2 23520.462} C_VEL
LIN {X 0,Y 290.253,Z 1146.204,A -85,B 0,C 180,E1 23530.416,E2 23530.416} C_VEL
LIN {X 0,Y 309.728,Z 1123.733,A -85,B 0,C 180,E1 23538.423,E2 23538.423} C_VEL
LIN {X 0,Y 333.771,Z 1094.498,A -85,B 0,C 180,E1 23545.453,E2 23545.453} C_VEL
LIN {X 0,Y 358.507,Z 1061.707,A -85,B 0,C 180,E1 23550.906,E2 23550.906} C_VEL
LIN {X 0,Y 382.907,Z 1024.571,A -85,B 0,C 180,E1 23555.189,E2 23555.189} C_VEL
LIN {X 0,Y 405.22,Z 984.51,A -85,B 0,C 180,E1 23558.53,E2 23558.53} C_VEL
LIN {X 0,Y 404.224,Z 967.761,A -85,B 0,C 180,E1 23563.746,E2 23563.746} C_VEL
LIN {X 0,Y 402.828,Z 955.292,A -85,B 0,C 180,E1 23569.203,E2 23569.203} C_VEL
LIN {X 0,Y 402.026,Z 947.714,A -85,B 0,C 180,E1 23574.621,E2 23574.621} C_VEL
LIN {X 0,Y 402.429,Z 944.672,A -85,B 0,C 180,E1 23577.861,E2 23577.861} C_VEL
LIN {X 0,Y 402.768,Z 943.934,A -85,B 0,C 180,E1 23580.012,E2 23580.012} C_VEL
LIN {X 0,Y 403.285,Z 949.573,A -85,B 0,C 180,E1 23586.466,E2 23586.466} C_VEL
LIN {X 0,Y 405.422,Z 959.186,A -85,B 0,C 180,E1 23592.033,E2 23592.033} C_VEL
LIN {X 0,Y 407.698,Z 973.317,A -85,B 0,C 180,E1 23597.259,E2 23597.259} C_VEL
LIN {X 0,Y 408.844,Z 983.731,A -85,B 0,C 180,E1 23600.256,E2 23600.256} C_VEL
LIN {X 0,Y 385.246,Z 1028.295,A -85,B 0,C 180,E1 23603.57,E2 23603.57} C_VEL
LIN {X 0,Y 360.235,Z 1067.552,A -85,B 0,C 180,E1 23607.779,E2 23607.779} C_VEL
LIN {X 0,Y 335.766,Z 1101.56,A -85,B 0,C 180,E1 23612.958,E2 23612.958} C_VEL
LIN {X 0,Y 310.735,Z 1133.144,A -85,B 0,C 180,E1 23620.008,E2 23620.008} C_VEL
LIN {X 0,Y 291.506,Z 1156.797,A -85,B 0,C 180,E1 23627.63,E2 23627.63} C_VEL
LIN {X 0,Y 276.313,Z 1176.281,A -85,B 0,C 180,E1 23636.845,E2 23636.845} C_VEL
LIN {X 0,Y 267.065,Z 1190.331,A -85,B 0,C 180,E1 23646.665,E2 23646.665} C_VEL
LIN {X 0,Y 262.993,Z 1199.319,A -85,B 0,C 180,E1 23656.711,E2 23656.711} C_VEL
LIN {X 0,Y 262.17,Z 1203.271,A -85,B 0,C 180,E1 23666.694,E2 23666.694} C_VEL
LIN {X 0,Y 262.282,Z 1203.277,A -85,B 0,C 180,E1 23673.301,E2 23673.301} C_VEL
LIN {X 0,Y 262.989,Z 1199.333,A -85,B 0,C 180,E1 23683.286,E2 23683.286} C_VEL
LIN {X 0,Y 267.072,Z 1190.359,A -85,B 0,C 180,E1 23693.331,E2 23693.331} C_VEL
LIN {X 0,Y 277.262,Z 1175.082,A -85,B 0,C 180,E1 23703.87,E2 23703.87} C_VEL
LIN {X 0,Y 292.638,Z 1155.483,A -85,B 0,C 180,E1 23712.862,E2 23712.862} C_VEL
LIN {X 0,Y 315.326,Z 1127.653,A -85,B 0,C 180,E1 23721.451,E2 23721.451} C_VEL
LIN {X 0,Y 339.164,Z 1097.089,A -85,B 0,C 180,E1 23727.833,E2 23727.833} C_VEL
LIN {X 0,Y 365.005,Z 1060.741,A -85,B 0,C 180,E1 23733.097,E2 23733.097} C_VEL
LIN {X 0,Y 389.417,Z 1021.103,A -85,B 0,C 180,E1 23737.058,E2 23737.058} C_VEL
LIN {X 0,Y 408.924,Z 983.897,A -85,B 0,C 180,E1 23739.745,E2 23739.745} C_VEL
LIN {X 0,Y 406.771,Z 967.023,A -85,B 0,C 180,E1 23744.917,E2 23744.917} C_VEL
LIN {X 0,Y 404.511,Z 954.769,A -85,B 0,C 180,E1 23750.311,E2 23750.311} C_VEL
LIN {X 0,Y 402.865,Z 947.563,A -85,B 0,C 180,E1 23755.686,E2 23755.686} C_VEL
LIN {X 0,Y 402.959,Z 944.112,A -85,B 0,C 180,E1 23759.988,E2 23759.988} C_VEL
LIN {X 0,Y 402.214,Z 947.956,A -85,B 0,C 180,E1 23765.376,E2 23765.376} C_VEL
LIN {X 0,Y 402.971,Z 955.641,A -85,B 0,C 180,E1 23770.793,E2 23770.793} C_VEL
LIN {X 0,Y 403.183,Z 957.423,A -85,B 0,C 180,E1 23771.75,E2 23771.75} C_VEL
LIN {X 0,Y 402.385,Z 963.125,A -85,B 0,C 180,E1 23773.427,E2 23773.427} C_VEL
LIN {X 0,Y 400.028,Z 974.664,A -85,B 0,C 180,E1 23776.113,E2 23776.113} C_VEL
LIN {X 0,Y 400.422,Z 988.909,A -85,B 0,C 180,E1 23780.64,E2 23780.64} C_VEL
LIN {X 0,Y 376.559,Z 1029.912,A -85,B 0,C 180,E1 23784.087,E2 23784.087} C_VEL
LIN {X 0,Y 351.438,Z 1066.368,A -85,B 0,C 180,E1 23788.45,E2 23788.45} C_VEL
LIN {X 0,Y 324.878,Z 1100.184,A -85,B 0,C 180,E1 23794.352,E2 23794.352} C_VEL
LIN {X 0,Y 301.552,Z 1127.09,A -85,B 0,C 180,E1 23801.267,E2 23801.267} C_VEL
LIN {X 0,Y 280.339,Z 1150.844,A -85,B 0,C 180,E1 23810.352,E2 23810.352} C_VEL
LIN {X 0,Y 265.91,Z 1167.497,A -85,B 0,C 180,E1 23820.184,E2 23820.184} C_VEL
LIN {X 0,Y 258.446,Z 1177.763,A -85,B 0,C 180,E1 23829.465,E2 23829.465} C_VEL
LIN {X 0,Y 254.768,Z 1184.444,A -85,B 0,C 180,E1 23839.752,E2 23839.752} C_VEL
LIN {X 0,Y 254.473,Z 1186.663,A -85,B 0,C 180,E1 23850.002,E2 23850.002} C_VEL
LIN {X 0,Y 254.834,Z 1184.385,A -85,B 0,C 180,E1 23860.249,E2 23860.249} C_VEL
LIN {X 0,Y 258.477,Z 1177.661,A -85,B 0,C 180,E1 23870.536,E2 23870.536} C_VEL
LIN {X 0,Y 266.978,Z 1166.239,A -85,B 0,C 180,E1 23880.626,E2 23880.626} C_VEL
LIN {X 0,Y 281.337,Z 1149.534,A -85,B 0,C 180,E1 23890.133,E2 23890.133} C_VEL
LIN {X 0,Y 302.718,Z 1125.744,A -85,B 0,C 180,E1 23899.041,E2 23899.041} C_VEL
LIN {X 0,Y 326.19,Z 1098.405,A -85,B 0,C 180,E1 23905.904,E2 23905.904} C_VEL
LIN {X 0,Y 352.244,Z 1065.174,A -85,B 0,C 180,E1 23911.607,E2 23911.607} C_VEL
LIN {X 0,Y 376.729,Z 1029.388,A -85,B 0,C 180,E1 23915.86,E2 23915.86} C_VEL
LIN {X 0,Y 400.286,Z 988.507,A -85,B 0,C 180,E1 23919.361,E2 23919.361} C_VEL
LIN {X 0,Y 399.731,Z 972.299,A -85,B 0,C 180,E1 23924.67,E2 23924.67} C_VEL
LIN {X 0,Y 398.71,Z 960.59,A -85,B 0,C 180,E1 23930.204,E2 23930.204} C_VEL
LIN {X 0,Y 398.451,Z 953.881,A -85,B 0,C 180,E1 23935.663,E2 23935.663} C_VEL
LIN {X 0,Y 399.25,Z 951.005,A -85,B 0,C 180,E1 23940.013,E2 23940.013} C_VEL
LIN {X 0,Y 399.71,Z 956.774,A -85,B 0,C 180,E1 23946.524,E2 23946.524} C_VEL
LIN {X 0,Y 401.294,Z 965.601,A -85,B 0,C 180,E1 23951.742,E2 23951.742} C_VEL
LIN {X 0,Y 403.219,Z 979.257,A -85,B 0,C 180,E1 23956.895,E2 23956.895} C_VEL
LIN {X 0,Y 403.735,Z 988.48,A -85,B 0,C 180,E1 23959.534,E2 23959.534} C_VEL
LIN {X 0,Y 381.005,Z 1029.703,A -85,B 0,C 180,E1 23962.6,E2 23962.6} C_VEL
LIN {X 0,Y 355.488,Z 1068.694,A -85,B 0,C 180,E1 23966.787,E2 23966.787} C_VEL
LIN {X 0,Y 330.745,Z 1102.006,A -85,B 0,C 180,E1 23971.892,E2 23971.892} C_VEL
LIN {X 0,Y 305.414,Z 1132.866,A -85,B 0,C 180,E1 23978.804,E2 23978.804} C_VEL
LIN {X 0,Y 285.417,Z 1156.522,A -85,B 0,C 180,E1 23986.504,E2 23986.504} C_VEL
LIN {X 0,Y 268.549,Z 1177.115,A -85,B 0,C 180,E1 23996.537,E2 23996.537} C_VEL
LIN {X 0,Y 259.572,Z 1190.061,A -85,B 0,C 180,E1 24005.95,E2 24005.95} C_VEL
LIN {X 0,Y 255.583,Z 1197.813,A -85,B 0,C 180,E1 24014.568,E2 24014.568} C_VEL
LIN {X 0,Y 254.225,Z 1202.17,A -85,B 0,C 180,E1 24023.171,E2 24023.171} C_VEL
LIN {X 0,Y 254.535,Z 1203.371,A -85,B 0,C 180,E1 24029.998,E2 24029.998} C_VEL
LIN {X 0,Y 254.235,Z 1202.178,A -85,B 0,C 180,E1 24036.825,E2 24036.825} C_VEL
LIN {X 0,Y 255.576,Z 1197.832,A -85,B 0,C 180,E1 24045.429,E2 24045.429} C_VEL
LIN {X 0,Y 260.427,Z 1188.657,A -85,B 0,C 180,E1 24055.278,E2 24055.278} C_VEL
LIN {X 0,Y 271.3,Z 1173.731,A -85,B 0,C 180,E1 24065.485,E2 24065.485} C_VEL
LIN {X 0,Y 288.605,Z 1152.806,A -85,B 0,C 180,E1 24074.876,E2 24074.876} C_VEL
LIN {X 0,Y 311.665,Z 1125.714,A -85,B 0,C 180,E1 24083.083,E2 24083.083} C_VEL
LIN {X 0,Y 337.264,Z 1093.638,A -85,B 0,C 180,E1 24089.572,E2 24089.572} C_VEL
LIN {X 0,Y 362.897,Z 1058.302,A -85,B 0,C 180,E1 24094.502,E2 24094.502} C_VEL
LIN {X 0,Y 388.507,Z 1017.1,A -85,B 0,C 180,E1 24098.467,E2 24098.467} C_VEL
LIN {X 0,Y 404.006,Z 988.01,A -85,B 0,C 180,E1 24100.554,E2 24100.554} C_VEL
LIN {X 0,Y 402.499,Z 973.247,A -85,B 0,C 180,E1 24105.253,E2 24105.253} C_VEL
LIN {X 0,Y 400.689,Z 962.015,A -85,B 0,C 180,E1 24110.218,E2 24110.218} C_VEL
LIN {X 0,Y 399.332,Z 954.686,A -85,B 0,C 180,E1 24115.648,E2 24115.648} C_VEL
LIN {X 0,Y 399.427,Z 951.21,A -85,B 0,C 180,E1 24119.987,E2 24119.987} C_VEL
LIN {X 0,Y 398.611,Z 955.083,A -85,B 0,C 180,E1 24125.425,E2 24125.425} C_VEL
LIN {X 0,Y 399.037,Z 962.854,A -85,B 0,C 180,E1 24130.9,E2 24130.9} C_VEL
LIN {X 0,Y 400.028,Z 974.664,A -85,B 0,C 180,E1 24136.113,E2 24136.113} C_VEL
LIN {X 0,Y 397.993,Z 981.823,A -85,B 0,C 180,E1 24137.419,E2 24137.419} C_VEL
LIN {X 0,Y 395.648,Z 989.355,A -85,B 0,C 180,E1 24138.715,E2 24138.715} C_VEL
LIN {X 0,Y 394.924,Z 994.14,A -85,B 0,C 180,E1 24139.915,E2 24139.915} C_VEL
LIN {X 0,Y 371.181,Z 1033.583,A -85,B 0,C 180,E1 24143.29,E2 24143.29} C_VEL
LIN {X 0,Y 345.844,Z 1068.934,A -85,B 0,C 180,E1 24147.604,E2 24147.604} C_VEL
LIN {X 0,Y 319.136,Z 1101.879,A -85,B 0,C 180,E1 24153.434,E2 24153.434} C_VEL
LIN {X 0,Y 294.21,Z 1129.479,A -85,B 0,C 180,E1 24160.751,E2 24160.751} C_VEL
LIN {X 0,Y 273.55,Z 1151.656,A -85,B 0,C 180,E1 24169.517,E2 24169.517} C_VEL
LIN {X 0,Y 257.891,Z 1168.874,A -85,B 0,C 180,E1 24180.13,E2 24180.13} C_VEL
LIN {X 0,Y 249.927,Z 1179.531,A -85,B 0,C 180,E1 24190.579,E2 24190.579} C_VEL
LIN {X 0,Y 246.916,Z 1184.706,A -85,B 0,C 180,E1 24199.422,E2 24199.422} C_VEL
LIN {X 0,Y 246.571,Z 1186.922,A -85,B 0,C 180,E1 24210.002,E2 24210.002} C_VEL
LIN {X 0,Y 246.979,Z 1184.647,A -85,B 0,C 180,E1 24220.578,E2 24220.578} C_VEL
LIN {X 0,Y 250.927,Z 1177.927,A -85,B 0,C 180,E1 24231.184,E2 24231.184} C_VEL
LIN {X 0,Y 259.95,Z 1166.509,A -85,B 0,C 180,E1 24241.548,E2 24241.548} C_VEL
LIN {X 0,Y 275.104,Z 1149.806,A -85,B 0,C 180,E1 24251.237,E2 24251.237} C_VEL
LIN {X 0,Y 297.383,Z 1126.017,A -85,B 0,C 180,E1 24260.24,E2 24260.24} C_VEL
LIN {X 0,Y 321.672,Z 1098.677,A -85,B 0,C 180,E1 24267.112,E2 24267.112} C_VEL
LIN {X 0,Y 349.02,Z 1064.708,A -85,B 0,C 180,E1 24272.891,E2 24272.891} C_VEL
LIN {X 0,Y 374.228,Z 1028.52,A -85,B 0,C 180,E1 24277.098,E2 24277.098} C_VEL
LIN {X 0,Y 395.392,Z 992.596,A -85,B 0,C 180,E1 24280.182,E2 24280.182} C_VEL
LIN {X 0,Y 395.3,Z 978.637,A -85,B 0,C 180,E1 24284.904,E2 24284.904} C_VEL
LIN {X 0,Y 394.761,Z 967.804,A -85,B 0,C 180,E1 24290.105,E2 24290.105} C_VEL
LIN {X 0,Y 394.596,Z 960.869,A -85,B 0,C 180,E1 24295.621,E2 24295.621} C_VEL
LIN {X 0,Y 395.58,Z 958.036,A -85,B 0,C 180,E1 24300.013,E2 24300.013} C_VEL
LIN {X 0,Y 395.917,Z 964.5,A -85,B 0,C 180,E1 24307.082,E2 24307.082} C_VEL
LIN {X 0,Y 397.526,Z 974.447,A -85,B 0,C 180,E1 24312.524,E2 24312.524} C_VEL
LIN {X 0,Y 398.894,Z 988.636,A -85,B 0,C 180,E1 24317.652,E2 24317.652} C_VEL
LIN {X 0,Y 398.88,Z 992.646,A -85,B 0,C 180,E1 24318.717,E2 24318.717} C_VEL
LIN {X 0,Y 374.643,Z 1034.577,A -85,B 0,C 180,E1 24321.918,E2 24321.918} C_VEL
LIN {X 0,Y 349.109,Z 1072.3,A -85,B 0,C 180,E1 24326.08,E2 24326.08} C_VEL
LIN {X 0,Y 323.669,Z 1105.016,A -85,B 0,C 180,E1 24331.279,E2 24331.279} C_VEL
LIN {X 0,Y 297.215,Z 1136.264,A -85,B 0,C 180,E1 24338.581,E2 24338.581} C_VEL
LIN {X 0,Y 275.126,Z 1160.974,A -85,B 0,C 180,E1 24347.341,E2 24347.341} C_VEL
LIN {X 0,Y 259.39,Z 1179.82,A -85,B 0,C 180,E1 24357.367,E2 24357.367} C_VEL
LIN {X 0,Y 249.981,Z 1193.29,A -85,B 0,C 180,E1 24368.732,E2 24368.732} C_VEL
LIN {X 0,Y 246.729,Z 1200.171,A -85,B 0,C 180,E1 24378.569,E2 24378.569} C_VEL
LIN {X 0,Y 246.36,Z 1202.751,A -85,B 0,C 180,E1 24386.482,E2 24386.482} C_VEL
LIN {X 0,Y 246.454,Z 1202.756,A -85,B 0,C 180,E1 24393.513,E2 24393.513} C_VEL
LIN {X 0,Y 247.357,Z 1198.806,A -85,B 0,C 180,E1 24404.142,E2 24404.142} C_VEL
LIN {X 0,Y 250.973,Z 1191.689,A -85,B 0,C 180,E1 24413.038,E2 24413.038} C_VEL
LIN {X 0,Y 260.982,Z 1177.799,A -85,B 0,C 180,E1 24423.902,E2 24423.902} C_VEL
LIN {X 0,Y 277.816,Z 1158.1,A -85,B 0,C 180,E1 24433.906,E2 24433.906} C_VEL
LIN {X 0,Y 299.212,Z 1133.909,A -85,B 0,C 180,E1 24442.1,E2 24442.1} C_VEL
LIN {X 0,Y 325.889,Z 1102.48,A -85,B 0,C 180,E1 24449.229,E2 24449.229} C_VEL
LIN {X 0,Y 351.832,Z 1068.601,A -85,B 0,C 180,E1 24454.412,E2 24454.412} C_VEL
LIN {X 0,Y 379.023,Z 1027.945,A -85,B 0,C 180,E1 24458.7,E2 24458.7} C_VEL
LIN {X 0,Y 398.921,Z 992.985,A -85,B 0,C 180,E1 24461.259,E2 24461.259} C_VEL
LIN {X 0,Y 398.224,Z 980.54,A -85,B 0,C 180,E1 24465.148,E2 24465.148} C_VEL
LIN {X 0,Y 396.77,Z 969.178,A -85,B 0,C 180,E1 24470.12,E2 24470.12} C_VEL
LIN {X 0,Y 395.535,Z 961.686,A -85,B 0,C 180,E1 24475.606,E2 24475.606} C_VEL
LIN {X 0,Y 395.746,Z 958.242,A -85,B 0,C 180,E1 24479.987,E2 24479.987} C_VEL
LIN {X 0,Y 394.738,Z 962.169,A -85,B 0,C 180,E1 24485.56,E2 24485.56} C_VEL
LIN {X 0,Y 395.14,Z 971.141,A -85,B 0,C 180,E1 24491.568,E2 24491.568} C_VEL
LIN {X 0,Y 395.667,Z 984.055,A -85,B 0,C 180,E1 24496.97,E2 24496.97} C_VEL
LIN {X 0,Y 395.648,Z 989.355,A -85,B 0,C 180,E1 24498.715,E2 24498.715} C_VEL
LIN {X 0,Y 393.528,Z 994.278,A -85,B 0,C 180,E1 24499.34,E2 24499.34} C_VEL
LIN {X 0,Y 384.056,Z 1008.508,A -85,B 0,C 180,E1 24499.858,E2 24499.858} C_VEL
LIN {X 0,Y 358.479,Z 1047.563,A -85,B 0,C 180,E1 24503.608,E2 24503.608} C_VEL
LIN {X 0,Y 332.478,Z 1081.268,A -85,B 0,C 180,E1 24508.269,E2 24508.269} C_VEL
LIN {X 0,Y 305.106,Z 1112.741,A -85,B 0,C 180,E1 24514.663,E2 24514.663} C_VEL
LIN {X 0,Y 280.865,Z 1138.022,A -85,B 0,C 180,E1 24522.406,E2 24522.406} C_VEL
LIN {X 0,Y 260.07,Z 1159.36,A -85,B 0,C 180,E1 24532.406,E2 24532.406} C_VEL
LIN {X 0,Y 247.008,Z 1173.638,A -85,B 0,C 180,E1 24543.139,E2 24543.139} C_VEL
LIN {X 0,Y 240.653,Z 1182.198,A -85,B 0,C 180,E1 24553.589,E2 24553.589} C_VEL
LIN {X 0,Y 238.578,Z 1186.138,A -85,B 0,C 180,E1 24562.724,E2 24562.724} C_VEL
LIN {X 0,Y 238.677,Z 1187.181,A -85,B 0,C 180,E1 24570.002,E2 24570.002} C_VEL
LIN {X 0,Y 239.159,Z 1184.909,A -85,B 0,C 180,E1 24580.929,E2 24580.929} C_VEL
LIN {X 0,Y 243.397,Z 1178.194,A -85,B 0,C 180,E1 24591.872,E2 24591.872} C_VEL
LIN {X 0,Y 253.02,Z 1166.778,A -85,B 0,C 180,E1 24602.516,E2 24602.516} C_VEL
LIN {X 0,Y 268.991,Z 1150.077,A -85,B 0,C 180,E1 24612.388,E2 24612.388} C_VEL
LIN {X 0,Y 292.707,Z 1125.773,A -85,B 0,C 180,E1 24621.642,E2 24621.642} C_VEL
LIN {X 0,Y 317.968,Z 1098.183,A -85,B 0,C 180,E1 24628.505,E2 24628.505} C_VEL
LIN {X 0,Y 345.21,Z 1065.203,A -85,B 0,C 180,E1 24634.06,E2 24634.06} C_VEL
LIN {X 0,Y 371.158,Z 1028.789,A -85,B 0,C 180,E1 24638.248,E2 24638.248} C_VEL
LIN {X 0,Y 390.544,Z 996.794,A -85,B 0,C 180,E1 24641.003,E2 24641.003} C_VEL
LIN {X 0,Y 390.795,Z 983.26,A -85,B 0,C 180,E1 24645.865,E2 24645.865} C_VEL
LIN {X 0,Y 390.643,Z 973.094,A -85,B 0,C 180,E1 24651.113,E2 24651.113} C_VEL
LIN {X 0,Y 391.244,Z 965.855,A -85,B 0,C 180,E1 24657.8,E2 24657.8} C_VEL
LIN {X 0,Y 391.734,Z 964.959,A -85,B 0,C 180,E1 24660.013,E2 24660.013} C_VEL
LIN {X 0,Y 391.921,Z 970.894,A -85,B 0,C 180,E1 24666.654,E2 24666.654} C_VEL
LIN {X 0,Y 393.144,Z 980.673,A -85,B 0,C 180,E1 24672.216,E2 24672.216} C_VEL
LIN {X 0,Y 394.21,Z 994.173,A -85,B 0,C 180,E1 24677.195,E2 24677.195} C_VEL
LIN {X 0,Y 394.22,Z 996.366,A -85,B 0,C 180,E1 24677.869,E2 24677.869} C_VEL
LIN {X 0,Y 368.005,Z 1039.992,A -85,B 0,C 180,E1 24681.269,E2 24681.269} C_VEL
LIN {X 0,Y 342.747,Z 1075.678,A -85,B 0,C 180,E1 24685.334,E2 24685.334} C_VEL
LIN {X 0,Y 315.305,Z 1109.646,A -85,B 0,C 180,E1 24690.967,E2 24690.967} C_VEL
LIN {X 0,Y 289.969,Z 1138.242,A -85,B 0,C 180,E1 24697.989,E2 24697.989} C_VEL
LIN {X 0,Y 266.266,Z 1163.882,A -85,B 0,C 180,E1 24707.562,E2 24707.562} C_VEL
LIN {X 0,Y 250.286,Z 1182.091,A -85,B 0,C 180,E1 24718.225,E2 24718.225} C_VEL
LIN {X 0,Y 241.513,Z 1194.627,A -85,B 0,C 180,E1 24729.847,E2 24729.847} C_VEL
LIN {X 0,Y 238.778,Z 1200.332,A -85,B 0,C 180,E1 24739.054,E2 24739.054} C_VEL
LIN {X 0,Y 238.444,Z 1202.49,A -85,B 0,C 180,E1 24746.365,E2 24746.365} C_VEL
LIN {X 0,Y 238.744,Z 1202.852,A -85,B 0,C 180,E1 24749.998,E2 24749.998} C_VEL
LIN {X 0,Y 238.446,Z 1201.657,A -85,B 0,C 180,E1 24757.28,E2 24757.28} C_VEL
LIN {X 0,Y 240.031,Z 1197.302,A -85,B 0,C 180,E1 24766.455,E2 24766.455} C_VEL
LIN {X 0,Y 246.018,Z 1187.624,A -85,B 0,C 180,E1 24777.365,E2 24777.365} C_VEL
LIN {X 0,Y 258.978,Z 1172.058,A -85,B 0,C 180,E1 24788.271,E2 24788.271} C_VEL
LIN {X 0,Y 279.78,Z 1149.248,A -85,B 0,C 180,E1 24798.439,E2 24798.439} C_VEL
LIN {X 0,Y 303.142,Z 1123.73,A -85,B 0,C 180,E1 24805.966,E2 24805.966} C_VEL
LIN {X 0,Y 331.49,Z 1090.249,A -85,B 0,C 180,E1 24812.536,E2 24812.536} C_VEL
LIN {X 0,Y 357.714,Z 1055.465,A -85,B 0,C 180,E1 24817.134,E2 24817.134} C_VEL
LIN {X 0,Y 383.149,Z 1016.063,A -85,B 0,C 180,E1 24820.77,E2 24820.77} C_VEL
LIN {X 0,Y 394.289,Z 996.546,A -85,B 0,C 180,E1 24822.135,E2 24822.135} C_VEL
LIN {X 0,Y 393.323,Z 982.215,A -85,B 0,C 180,E1 24827.226,E2 24827.226} C_VEL
LIN {X 0,Y 392.189,Z 972.113,A -85,B 0,C 180,E1 24832.621,E2 24832.621} C_VEL
LIN {X 0,Y 391.892,Z 965.181,A -85,B 0,C 180,E1 24839.987,E2 24839.987} C_VEL
LIN {X 0,Y 390.867,Z 969.175,A -85,B 0,C 180,E1 24845.615,E2 24845.615} C_VEL
LIN {X 0,Y 390.87,Z 978.416,A -85,B 0,C 180,E1 24851.794,E2 24851.794} C_VEL
LIN {X 0,Y 390.97,Z 990.702,A -85,B 0,C 180,E1 24856.89,E2 24856.89} C_VEL
LIN {X 0,Y 390.385,Z 997.722,A -85,B 0,C 180,E1 24859.041,E2 24859.041} C_VEL
LIN {X 0,Y 384.056,Z 1008.508,A -85,B 0,C 180,E1 24859.858,E2 24859.858} C_VEL
LIN {X 0,Y 374.098,Z 1022.448,A -85,B 0,C 180,E1 24860.444,E2 24860.444} C_VEL
LIN {X 0,Y 363.831,Z 1035.884,A -85,B 0,C 180,E1 24861.136,E2 24861.136} C_VEL
LIN {X 0,Y 335.469,Z 1073.353,A -85,B 0,C 180,E1 24865.727,E2 24865.727} C_VEL
LIN {X 0,Y 308.104,Z 1104.813,A -85,B 0,C 180,E1 24871.441,E2 24871.441} C_VEL
LIN {X 0,Y 280.642,Z 1133.195,A -85,B 0,C 180,E1 24879.286,E2 24879.286} C_VEL
LIN {X 0,Y 259.597,Z 1153.703,A -85,B 0,C 180,E1 24887.98,E2 24887.98} C_VEL
LIN {X 0,Y 242.834,Z 1170.517,A -85,B 0,C 180,E1 24899.113,E2 24899.113} C_VEL
LIN {X 0,Y 234.473,Z 1180.461,A -85,B 0,C 180,E1 24909.779,E2 24909.779} C_VEL
LIN {X 0,Y 231.266,Z 1185.228,A -85,B 0,C 180,E1 24918.697,E2 24918.697} C_VEL
LIN {X 0,Y 230.773,Z 1187.441,A -85,B 0,C 180,E1 24930.002,E2 24930.002} C_VEL
LIN {X 0,Y 231.315,Z 1185.172,A -85,B 0,C 180,E1 24941.304,E2 24941.304} C_VEL
LIN {X 0,Y 235.89,Z 1178.461,A -85,B 0,C 180,E1 24952.606,E2 24952.606} C_VEL
LIN {X 0,Y 246.146,Z 1167.048,A -85,B 0,C 180,E1 24963.542,E2 24963.542} C_VEL
LIN {X 0,Y 262.981,Z 1150.348,A -85,B 0,C 180,E1 24973.595,E2 24973.595} C_VEL
LIN {X 0,Y 287.233,Z 1126.49,A -85,B 0,C 180,E1 24982.781,E2 24982.781} C_VEL
LIN {X 0,Y 312.83,Z 1099.51,A -85,B 0,C 180,E1 24989.569,E2 24989.569} C_VEL
LIN {X 0,Y 341.737,Z 1065.473,A -85,B 0,C 180,E1 24995.284,E2 24995.284} C_VEL
LIN {X 0,Y 367.27,Z 1030.534,A -85,B 0,C 180,E1 24999.275,E2 24999.275} C_VEL
LIN {X 0,Y 385.759,Z 1001.285,A -85,B 0,C 180,E1 25001.753,E2 25001.753} C_VEL
LIN {X 0,Y 386.314,Z 988.797,A -85,B 0,C 180,E1 25006.441,E2 25006.441} C_VEL
LIN {X 0,Y 386.45,Z 978.419,A -85,B 0,C 180,E1 25012.148,E2 25012.148} C_VEL
LIN {X 0,Y 387.34,Z 972.834,A -85,B 0,C 180,E1 25017.777,E2 25017.777} C_VEL
LIN {X 0,Y 387.889,Z 971.88,A -85,B 0,C 180,E1 25020.013,E2 25020.013} C_VEL
LIN {X 0,Y 387.854,Z 977.878,A -85,B 0,C 180,E1 25026.724,E2 25026.724} C_VEL
LIN {X 0,Y 388.697,Z 986.619,A -85,B 0,C 180,E1 25031.789,E2 25031.789} C_VEL
LIN {X 0,Y 389.333,Z 1000.024,A -85,B 0,C 180,E1 25036.892,E2 25036.892} C_VEL
LIN {X 0,Y 363.342,Z 1042.442,A -85,B 0,C 180,E1 25040.322,E2 25040.322} C_VEL
LIN {X 0,Y 334.907,Z 1080.881,A -85,B 0,C 180,E1 25044.829,E2 25044.829} C_VEL
LIN {X 0,Y 307.161,Z 1113.908,A -85,B 0,C 180,E1 25050.576,E2 25050.576} C_VEL
LIN {X 0,Y 280.012,Z 1143.071,A -85,B 0,C 180,E1 25058.276,E2 25058.276} C_VEL
LIN {X 0,Y 258.483,Z 1165.404,A -85,B 0,C 180,E1 25067.207,E2 25067.207} C_VEL
LIN {X 0,Y 242.213,Z 1183.102,A -85,B 0,C 180,E1 25078.18,E2 25078.18} C_VEL
LIN {X 0,Y 233.872,Z 1194.359,A -85,B 0,C 180,E1 25089.158,E2 25089.158} C_VEL
LIN {X 0,Y 230.852,Z 1200.293,A -85,B 0,C 180,E1 25099.15,E2 25099.15} C_VEL
LIN {X 0,Y 230.839,Z 1202.593,A -85,B 0,C 180,E1 25109.998,E2 25109.998} C_VEL
LIN {X 0,Y 230.541,Z 1201.395,A -85,B 0,C 180,E1 25117.531,E2 25117.531} C_VEL
LIN {X 0,Y 232.293,Z 1197.038,A -85,B 0,C 180,E1 25127.02,E2 25127.02} C_VEL
LIN {X 0,Y 239.013,Z 1187.06,A -85,B 0,C 180,E1 25138.543,E2 25138.543} C_VEL
LIN {X 0,Y 252.553,Z 1171.688,A -85,B 0,C 180,E1 25149.499,E2 25149.499} C_VEL
LIN {X 0,Y 273.656,Z 1149.657,A -85,B 0,C 180,E1 25159.488,E2 25159.488} C_VEL
LIN {X 0,Y 298.569,Z 1123.459,A -85,B 0,C 180,E1 25167.288,E2 25167.288} C_VEL
LIN {X 0,Y 328.042,Z 1089.611,A -85,B 0,C 180,E1 25173.887,E2 25173.887} C_VEL
LIN {X 0,Y 355.338,Z 1054.138,A -85,B 0,C 180,E1 25178.471,E2 25178.471} C_VEL
LIN {X 0,Y 381.291,Z 1014.603,A -85,B 0,C 180,E1 25182.015,E2 25182.015} C_VEL
LIN {X 0,Y 389.375,Z 1000.307,A -85,B 0,C 180,E1 25183.094,E2 25183.094} C_VEL
LIN {X 0,Y 388.771,Z 986.862,A -85,B 0,C 180,E1 25188.214,E2 25188.214} C_VEL
LIN {X 0,Y 387.983,Z 978.072,A -85,B 0,C 180,E1 25193.278,E2 25193.278} C_VEL
LIN {X 0,Y 388.044,Z 972.112,A -85,B 0,C 180,E1 25199.987,E2 25199.987} C_VEL
LIN {X 0,Y 386.794,Z 975.984,A -85,B 0,C 180,E1 25205.591,E2 25205.591} C_VEL
LIN {X 0,Y 386.528,Z 984.285,A -85,B 0,C 180,E1 25211.258,E2 25211.258} C_VEL
LIN {X 0,Y 386.207,Z 996.322,A -85,B 0,C 180,E1 25216.464,E2 25216.464} C_VEL
LIN {X 0,Y 385.443,Z 1002.206,A -85,B 0,C 180,E1 25218.216,E2 25218.216} C_VEL
LIN {X 0,Y 363.831,Z 1035.884,A -85,B 0,C 180,E1 25221.136,E2 25221.136} C_VEL
LIN {X 0,Y 352.995,Z 1049.031,A -85,B 0,C 180,E1 25221.91,E2 25221.91} C_VEL
LIN {X 0,Y 342.015,Z 1061.393,A -85,B 0,C 180,E1 25222.78,E2 25222.78} C_VEL
LIN {X 0,Y 314.098,Z 1094.166,A -85,B 0,C 180,E1 25227.913,E2 25227.913} C_VEL
LIN {X 0,Y 285.541,Z 1123.799,A -85,B 0,C 180,E1 25234.89,E2 25234.89} C_VEL
LIN {X 0,Y 260.835,Z 1147.153,A -85,B 0,C 180,E1 25243.397,E2 25243.397} C_VEL
LIN {X 0,Y 241.831,Z 1164.965,A -85,B 0,C 180,E1 25253.493,E2 25253.493} C_VEL
LIN {X 0,Y 229.761,Z 1177.325,A -85,B 0,C 180,E1 25264.693,E2 25264.693} C_VEL
LIN {X 0,Y 224.545,Z 1183.856,A -85,B 0,C 180,E1 25274.386,E2 25274.386} C_VEL
LIN {X 0,Y 222.639,Z 1187.396,A -85,B 0,C 180,E1 25286.11,E2 25286.11} C_VEL
LIN {X 0,Y 222.694,Z 1187.383,A -85,B 0,C 180,E1 25293.893,E2 25293.893} C_VEL
LIN {X 0,Y 224.573,Z 1183.796,A -85,B 0,C 180,E1 25305.616,E2 25305.616} C_VEL
LIN {X 0,Y 231.346,Z 1175.485,A -85,B 0,C 180,E1 25317.21,E2 25317.21} C_VEL
LIN {X 0,Y 246.698,Z 1160.334,A -85,B 0,C 180,E1 25329.501,E2 25329.501} C_VEL
LIN {X 0,Y 268.394,Z 1139.999,A -85,B 0,C 180,E1 25339.504,E2 25339.504} C_VEL
LIN {X 0,Y 295.274,Z 1113.994,A -85,B 0,C 180,E1 25347.665,E2 25347.665} C_VEL
LIN {X 0,Y 323.54,Z 1083.337,A -85,B 0,C 180,E1 25353.909,E2 25353.909} C_VEL
LIN {X 0,Y 350.791,Z 1049.892,A -85,B 0,C 180,E1 25358.519,E2 25358.519} C_VEL
LIN {X 0,Y 377.931,Z 1010.325,A -85,B 0,C 180,E1 25362.201,E2 25362.201} C_VEL
LIN {X 0,Y 380.275,Z 1006.58,A -85,B 0,C 180,E1 25362.5,E2 25362.5} C_VEL
LIN {X 0,Y 381.267,Z 1001.838,A -85,B 0,C 180,E1 25363.908,E2 25363.908} C_VEL
LIN {X 0,Y 381.959,Z 989.978,A -85,B 0,C 180,E1 25369.183,E2 25369.183} C_VEL
LIN {X 0,Y 382.4,Z 982.637,A -85,B 0,C 180,E1 25374.344,E2 25374.344} C_VEL
LIN {X 0,Y 383.766,Z 978.665,A -85,B 0,C 180,E1 25380.013,E2 25380.013} C_VEL
LIN {X 0,Y 383.623,Z 984.791,A -85,B 0,C 180,E1 25386.799,E2 25386.799} C_VEL
LIN {X 0,Y 384.321,Z 993.768,A -85,B 0,C 180,E1 25391.925,E2 25391.925} C_VEL
LIN {X 0,Y 384.435,Z 1004.132,A -85,B 0,C 180,E1 25395.983,E2 25395.983} C_VEL
LIN {X 0,Y 380.334,Z 1011.712,A -85,B 0,C 180,E1 25396.641,E2 25396.641} C_VEL
LIN {X 0,Y 353.491,Z 1052.098,A -85,B 0,C 180,E1 25400.111,E2 25400.111} C_VEL
LIN {X 0,Y 325.199,Z 1088.352,A -85,B 0,C 180,E1 25404.661,E2 25404.661} C_VEL
LIN {X 0,Y 294.959,Z 1122.181,A -85,B 0,C 180,E1 25411.136,E2 25411.136} C_VEL
LIN {X 0,Y 270.256,Z 1147.466,A -85,B 0,C 180,E1 25418.48,E2 25418.48} C_VEL
LIN {X 0,Y 247.42,Z 1170.098,A -85,B 0,C 180,E1 25428.584,E2 25428.584} C_VEL
LIN {X 0,Y 232.504,Z 1185.988,A -85,B 0,C 180,E1 25439.753,E2 25439.753} C_VEL
LIN {X 0,Y 225.346,Z 1195.487,A -85,B 0,C 180,E1 25450.408,E2 25450.408} C_VEL
LIN {X 0,Y 223.074,Z 1199.806,A -85,B 0,C 180,E1 25458.273,E2 25458.273} C_VEL
LIN {X 0,Y 222.63,Z 1201.97,A -85,B 0,C 180,E1 25466.106,E2 25466.106} C_VEL
LIN {X 0,Y 222.932,Z 1202.333,A -85,B 0,C 180,E1 25469.998,E2 25469.998} C_VEL
LIN {X 0,Y 222.646,Z 1201.134,A -85,B 0,C 180,E1 25477.8,E2 25477.8} C_VEL
LIN {X 0,Y 224.569,Z 1196.773,A -85,B 0,C 180,E1 25487.624,E2 25487.624} C_VEL
LIN {X 0,Y 231.617,Z 1187.022,A -85,B 0,C 180,E1 25499.293,E2 25499.293} C_VEL
LIN {X 0,Y 246.41,Z 1171.214,A -85,B 0,C 180,E1 25510.837,E2 25510.837} C_VEL
LIN {X 0,Y 268.162,Z 1149.534,A -85,B 0,C 180,E1 25520.786,E2 25520.786} C_VEL
LIN {X 0,Y 293.785,Z 1123.574,A -85,B 0,C 180,E1 25528.567,E2 25528.567} C_VEL
LIN {X 0,Y 323.638,Z 1090.308,A -85,B 0,C 180,E1 25535.049,E2 25535.049} C_VEL
LIN {X 0,Y 351.654,Z 1054.932,A -85,B 0,C 180,E1 25539.602,E2 25539.602} C_VEL
LIN {X 0,Y 377.952,Z 1015.791,A -85,B 0,C 180,E1 25543.076,E2 25543.076} C_VEL
LIN {X 0,Y 383.964,Z 1005.856,A -85,B 0,C 180,E1 25543.76,E2 25543.76} C_VEL
LIN {X 0,Y 384.529,Z 1000.993,A -85,B 0,C 180,E1 25545.189,E2 25545.189} C_VEL
LIN {X 0,Y 384.151,Z 989.692,A -85,B 0,C 180,E1 25550.206,E2 25550.206} C_VEL
LIN {X 0,Y 383.543,Z 982.41,A -85,B 0,C 180,E1 25555.468,E2 25555.468} C_VEL
LIN {X 0,Y 383.922,Z 978.874,A -85,B 0,C 180,E1 25559.987,E2 25559.987} C_VEL
LIN {X 0,Y 382.586,Z 982.847,A -85,B 0,C 180,E1 25565.653,E2 25565.653} C_VEL
LIN {X 0,Y 382.044,Z 991.324,A -85,B 0,C 180,E1 25571.392,E2 25571.392} C_VEL
LIN {X 0,Y 381.332,Z 1003.859,A -85,B 0,C 180,E1 25576.724,E2 25576.724} C_VEL
LIN {X 0,Y 381.16,Z 1005.241,A -85,B 0,C 180,E1 25577.21,E2 25577.21} C_VEL
LIN {X 0,Y 352.768,Z 1047.437,A -85,B 0,C 180,E1 25581.121,E2 25581.121} C_VEL
LIN {X 0,Y 342.015,Z 1061.393,A -85,B 0,C 180,E1 25582.78,E2 25582.78} C_VEL
LIN {X 0,Y 330.682,Z 1073.445,A -85,B 0,C 180,E1 25583.775,E2 25583.775} C_VEL
LIN {X 0,Y 319.031,Z 1084.916,A -85,B 0,C 180,E1 25584.889,E2 25584.889} C_VEL
LIN {X 0,Y 290.204,Z 1115.12,A -85,B 0,C 180,E1 25591.066,E2 25591.066} C_VEL
LIN {X 0,Y 262.699,Z 1140.776,A -85,B 0,C 180,E1 25599.223,E2 25599.223} C_VEL
LIN {X 0,Y 241.451,Z 1159.84,A -85,B 0,C 180,E1 25608.639,E2 25608.639} C_VEL
LIN {X 0,Y 225.093,Z 1174.809,A -85,B 0,C 180,E1 25620.718,E2 25620.718} C_VEL
LIN {X 0,Y 217.608,Z 1182.989,A -85,B 0,C 180,E1 25631.793,E2 25631.793} C_VEL
LIN {X 0,Y 214.926,Z 1186.921,A -85,B 0,C 180,E1 25641.918,E2 25641.918} C_VEL
LIN {X 0,Y 214.966,Z 1187.959,A -85,B 0,C 180,E1 25650.002,E2 25650.002} C_VEL
LIN {X 0,Y 215.67,Z 1185.697,A -85,B 0,C 180,E1 25662.136,E2 25662.136} C_VEL
LIN {X 0,Y 220.996,Z 1178.995,A -85,B 0,C 180,E1 25674.224,E2 25674.224} C_VEL
LIN {X 0,Y 233.364,Z 1166.976,A -85,B 0,C 180,E1 25686.283,E2 25686.283} C_VEL
LIN {X 0,Y 253.967,Z 1148.51,A -85,B 0,C 180,E1 25697.306,E2 25697.306} C_VEL
LIN {X 0,Y 279.867,Z 1124.977,A -85,B 0,C 180,E1 25706.118,E2 25706.118} C_VEL
LIN {X 0,Y 308.998,Z 1095.682,A -85,B 0,C 180,E1 25713.074,E2 25713.074} C_VEL
LIN {X 0,Y 337.749,Z 1062.982,A -85,B 0,C 180,E1 25718.211,E2 25718.211} C_VEL
LIN {X 0,Y 365.909,Z 1025.176,A -85,B 0,C 180,E1 25722.206,E2 25722.206} C_VEL
LIN {X 0,Y 376.103,Z 1009.522,A -85,B 0,C 180,E1 25723.526,E2 25723.526} C_VEL
LIN {X 0,Y 377.254,Z 997.996,A -85,B 0,C 180,E1 25728.462,E2 25728.462} C_VEL
LIN {X 0,Y 378.168,Z 989.479,A -85,B 0,C 180,E1 25734.281,E2 25734.281} C_VEL
LIN {X 0,Y 379.604,Z 985.417,A -85,B 0,C 180,E1 25740.013,E2 25740.013} C_VEL
LIN {X 0,Y 379.392,Z 991.687,A -85,B 0,C 180,E1 25746.875,E2 25746.875} C_VEL
LIN {X 0,Y 379.661,Z 1000.768,A -85,B 0,C 180,E1 25752.073,E2 25752.073} C_VEL
LIN {X 0,Y 379.617,Z 1008.746,A -85,B 0,C 180,E1 25755.224,E2 25755.224} C_VEL
LIN {X 0,Y 352.705,Z 1049.125,A -85,B 0,C 180,E1 25758.571,E2 25758.571} C_VEL
LIN {X 0,Y 324.017,Z 1085.557,A -85,B 0,C 180,E1 25762.943,E2 25762.943} C_VEL
LIN {X 0,Y 295.082,Z 1117.4,A -85,B 0,C 180,E1 25768.718,E2 25768.718} C_VEL
LIN {X 0,Y 266.646,Z 1145.84,A -85,B 0,C 180,E1 25776.58,E2 25776.58} C_VEL
LIN {X 0,Y 242.334,Z 1168.758,A -85,B 0,C 180,E1 25786.689,E2 25786.689} C_VEL
LIN {X 0,Y 226.42,Z 1184.693,A -85,B 0,C 180,E1 25797.728,E2 25797.728} C_VEL
LIN {X 0,Y 217.714,Z 1195.22,A -85,B 0,C 180,E1 25809.692,E2 25809.692} C_VEL
LIN {X 0,Y 214.858,Z 1200.357,A -85,B 0,C 180,E1 25820.035,E2 25820.035} C_VEL
LIN {X 0,Y 215.026,Z 1202.074,A -85,B 0,C 180,E1 25829.998,E2 25829.998} C_VEL
LIN {X 0,Y 214.887,Z 1200.354,A -85,B 0,C 180,E1 25840.009,E2 25840.009} C_VEL
LIN {X 0,Y 217.712,Z 1195.243,A -85,B 0,C 180,E1 25850.304,E2 25850.304} C_VEL
LIN {X 0,Y 226.441,Z 1184.738,A -85,B 0,C 180,E1 25862.265,E2 25862.265} C_VEL
LIN {X 0,Y 244.448,Z 1166.868,A -85,B 0,C 180,E1 25874.362,E2 25874.362} C_VEL
LIN {X 0,Y 268.231,Z 1144.376,A -85,B 0,C 180,E1 25883.926,E2 25883.926} C_VEL
LIN {X 0,Y 297.713,Z 1114.837,A -85,B 0,C 180,E1 25891.87,E2 25891.87} C_VEL
LIN {X 0,Y 325.569,Z 1083.915,A -85,B 0,C 180,E1 25897.287,E2 25897.287} C_VEL
LIN {X 0,Y 355.856,Z 1045.123,A -85,B 0,C 180,E1 25901.826,E2 25901.826} C_VEL
LIN {X 0,Y 379.083,Z 1010.187,A -85,B 0,C 180,E1 25904.636,E2 25904.636} C_VEL
LIN {X 0,Y 379.732,Z 1006.263,A -85,B 0,C 180,E1 25905.757,E2 25905.757} C_VEL
LIN {X 0,Y 379.62,Z 995.35,A -85,B 0,C 180,E1 25910.826,E2 25910.826} C_VEL
LIN {X 0,Y 379.309,Z 988.2,A -85,B 0,C 180,E1 25916.561,E2 25916.561} C_VEL
LIN {X 0,Y 379.755,Z 985.639,A -85,B 0,C 180,E1 25919.987,E2 25919.987} C_VEL
LIN {X 0,Y 378.337,Z 989.696,A -85,B 0,C 180,E1 25925.717,E2 25925.717} C_VEL
LIN {X 0,Y 377.395,Z 998.295,A -85,B 0,C 180,E1 25931.534,E2 25931.534} C_VEL
LIN {X 0,Y 376.36,Z 1009.308,A -85,B 0,C 180,E1 25936.307,E2 25936.307} C_VEL
LIN {X 0,Y 348.783,Z 1049.254,A -85,B 0,C 180,E1 25940.046,E2 25940.046} C_VEL
LIN {X 0,Y 320.134,Z 1083.683,A -85,B 0,C 180,E1 25944.684,E2 25944.684} C_VEL
LIN {X 0,Y 319.031,Z 1084.916,A -85,B 0,C 180,E1 25944.889,E2 25944.889} C_VEL
LIN {X 0,Y 307.234,Z 1095.962,A -85,B 0,C 180,E1 25946.146,E2 25946.146} C_VEL
LIN {X 0,Y 295.221,Z 1106.387,A -85,B 0,C 180,E1 25947.551,E2 25947.551} C_VEL
LIN {X 0,Y 265.608,Z 1134.04,A -85,B 0,C 180,E1 25955.16,E2 25955.16} C_VEL
LIN {X 0,Y 241.446,Z 1154.804,A -85,B 0,C 180,E1 25964.224,E2 25964.224} C_VEL
LIN {X 0,Y 222.997,Z 1170.572,A -85,B 0,C 180,E1 25975.222,E2 25975.222} C_VEL
LIN {X 0,Y 211.458,Z 1181.644,A -85,B 0,C 180,E1 25988.197,E2 25988.197} C_VEL
LIN {X 0,Y 207.821,Z 1186.014,A -85,B 0,C 180,E1 25997.403,E2 25997.403} C_VEL
LIN {X 0,Y 207.065,Z 1188.219,A -85,B 0,C 180,E1 26010.002,E2 26010.002} C_VEL
LIN {X 0,Y 207.117,Z 1187.148,A -85,B 0,C 180,E1 26018.393,E2 26018.393} C_VEL
LIN {X 0,Y 209.99,Z 1183.179,A -85,B 0,C 180,E1 26028.897,E2 26028.897} C_VEL
LIN {X 0,Y 219.635,Z 1173.59,A -85,B 0,C 180,E1 26041.789,E2 26041.789} C_VEL
LIN {X 0,Y 236.923,Z 1158.569,A -85,B 0,C 180,E1 26053.481,E2 26053.481} C_VEL
LIN {X 0,Y 262.42,Z 1136.786,A -85,B 0,C 180,E1 26063.726,E2 26063.726} C_VEL
LIN {X 0,Y 290.024,Z 1111.323,A -85,B 0,C 180,E1 26071.205,E2 26071.205} C_VEL
LIN {X 0,Y 319.891,Z 1080.458,A -85,B 0,C 180,E1 26077.098,E2 26077.098} C_VEL
LIN {X 0,Y 348.648,Z 1045.81,A -85,B 0,C 180,E1 26081.51,E2 26081.51} C_VEL
LIN {X 0,Y 371.33,Z 1013.621,A -85,B 0,C 180,E1 26084.472,E2 26084.472} C_VEL
LIN {X 0,Y 372.779,Z 1003.097,A -85,B 0,C 180,E1 26089.304,E2 26089.304} C_VEL
LIN {X 0,Y 373.656,Z 996.142,A -85,B 0,C 180,E1 26094.212,E2 26094.212} C_VEL
LIN {X 0,Y 375.356,Z 992.106,A -85,B 0,C 180,E1 26100.013,E2 26100.013} C_VEL
LIN {X 0,Y 374.858,Z 998.409,A -85,B 0,C 180,E1 26106.959,E2 26106.959} C_VEL
LIN {X 0,Y 374.984,Z 1006.499,A -85,B 0,C 180,E1 26111.636,E2 26111.636} C_VEL
LIN {X 0,Y 374.495,Z 1013.505,A -85,B 0,C 180,E1 26114.434,E2 26114.434} C_VEL
LIN {X 0,Y 346.594,Z 1053.691,A -85,B 0,C 180,E1 26117.783,E2 26117.783} C_VEL
LIN {X 0,Y 317.709,Z 1088.842,A -85,B 0,C 180,E1 26122.118,E2 26122.118} C_VEL
LIN {X 0,Y 286.512,Z 1121.867,A -85,B 0,C 180,E1 26128.354,E2 26128.354} C_VEL
LIN {X 0,Y 260.232,Z 1146.917,A -85,B 0,C 180,E1 26135.612,E2 26135.612} C_VEL
LIN {X 0,Y 234.654,Z 1170.057,A -85,B 0,C 180,E1 26146.187,E2 26146.187} C_VEL
LIN {X 0,Y 218.406,Z 1185.445,A -85,B 0,C 180,E1 26157.572,E2 26157.572} C_VEL
LIN {X 0,Y 209.869,Z 1195.267,A -85,B 0,C 180,E1 26169.444,E2 26169.444} C_VEL
LIN {X 0,Y 206.858,Z 1200.601,A -85,B 0,C 180,E1 26181.597,E2 26181.597} C_VEL
LIN {X 0,Y 207.13,Z 1201.815,A -85,B 0,C 180,E1 26189.998,E2 26189.998} C_VEL
LIN {X 0,Y 206.868,Z 1200.611,A -85,B 0,C 180,E1 26198.399,E2 26198.399} C_VEL
LIN {X 0,Y 209.885,Z 1195.281,A -85,B 0,C 180,E1 26210.567,E2 26210.567} C_VEL
LIN {X 0,Y 219.493,Z 1184.467,A -85,B 0,C 180,E1 26223.417,E2 26223.417} C_VEL
LIN {X 0,Y 238.69,Z 1166.463,A -85,B 0,C 180,E1 26235.839,E2 26235.839} C_VEL
LIN {X 0,Y 263.686,Z 1143.828,A -85,B 0,C 180,E1 26245.484,E2 26245.484} C_VEL
LIN {X 0,Y 293.874,Z 1114.565,A -85,B 0,C 180,E1 26253.304,E2 26253.304} C_VEL
LIN {X 0,Y 323.932,Z 1081.866,A -85,B 0,C 180,E1 26258.901,E2 26258.901} C_VEL
LIN {X 0,Y 354.973,Z 1042.735,A -85,B 0,C 180,E1 26263.295,E2 26263.295} C_VEL
LIN {X 0,Y 374.489,Z 1013.816,A -85,B 0,C 180,E1 26265.56,E2 26265.56} C_VEL
LIN {X 0,Y 375.023,Z 1004.369,A -85,B 0,C 180,E1 26269.541,E2 26269.541} C_VEL
LIN {X 0,Y 374.95,Z 996.699,A -85,B 0,C 180,E1 26274.607,E2 26274.607} C_VEL
LIN {X 0,Y 375.493,Z 992.328,A -85,B 0,C 180,E1 26279.987,E2 26279.987} C_VEL
LIN {X 0,Y 373.815,Z 996.374,A -85,B 0,C 180,E1 26285.786,E2 26285.786} C_VEL
LIN {X 0,Y 372.701,Z 1005.259,A -85,B 0,C 180,E1 26291.681,E2 26291.681} C_VEL
LIN {X 0,Y 371.624,Z 1013.088,A -85,B 0,C 180,E1 26295.223,E2 26295.223} C_VEL
LIN {X 0,Y 370.083,Z 1016.097,A -85,B 0,C 180,E1 26295.704,E2 26295.704} C_VEL
LIN {X 0,Y 343.443,Z 1052.805,A -85,B 0,C 180,E1 26299.148,E2 26299.148} C_VEL
LIN {X 0,Y 312.368,Z 1088.802,A -85,B 0,C 180,E1 26304.138,E2 26304.138} C_VEL
LIN {X 0,Y 295.221,Z 1106.387,A -85,B 0,C 180,E1 26307.551,E2 26307.551} C_VEL
LIN {X 0,Y 283.031,Z 1116.37,A -85,B 0,C 180,E1 26309.133,E2 26309.133} C_VEL
LIN {X 0,Y 271.035,Z 1125.643,A -85,B 0,C 180,E1 26310.913,E2 26310.913} C_VEL
LIN {X 0,Y 244.165,Z 1148.247,A -85,B 0,C 180,E1 26319.323,E2 26319.323} C_VEL
LIN {X 0,Y 220.871,Z 1167.158,A -85,B 0,C 180,E1 26330.742,E2 26330.742} C_VEL
LIN {X 0,Y 206.265,Z 1179.621,A -85,B 0,C 180,E1 26343.926,E2 26343.926} C_VEL
LIN {X 0,Y 200.023,Z 1186.276,A -85,B 0,C 180,E1 26356.903,E2 26356.903} C_VEL
LIN {X 0,Y 199.16,Z 1188.478,A -85,B 0,C 180,E1 26370.002,E2 26370.002} C_VEL
LIN {X 0,Y 199.392,Z 1187.118,A -85,B 0,C 180,E1 26380.051,E2 26380.051} C_VEL
LIN {X 0,Y 203.51,Z 1182.292,A -85,B 0,C 180,E1 26391.796,E2 26391.796} C_VEL
LIN {X 0,Y 214.367,Z 1172.556,A -85,B 0,C 180,E1 26404.331,E2 26404.331} C_VEL
LIN {X 0,Y 234.155,Z 1156.289,A -85,B 0,C 180,E1 26416.378,E2 26416.378} C_VEL
LIN {X 0,Y 259.261,Z 1135.728,A -85,B 0,C 180,E1 26425.708,E2 26425.708} C_VEL
LIN {X 0,Y 289.479,Z 1108.426,A -85,B 0,C 180,E1 26433.369,E2 26433.369} C_VEL
LIN {X 0,Y 319.801,Z 1077.493,A -85,B 0,C 180,E1 26438.946,E2 26438.946} C_VEL
LIN {X 0,Y 350.689,Z 1040.224,A -85,B 0,C 180,E1 26443.349,E2 26443.349} C_VEL
LIN {X 0,Y 366.613,Z 1017.875,A -85,B 0,C 180,E1 26445.393,E2 26445.393} C_VEL
LIN {X 0,Y 368.263,Z 1007.566,A -85,B 0,C 180,E1 26450.568,E2 26450.568} C_VEL
LIN {X 0,Y 369.394,Z 1001.666,A -85,B 0,C 180,E1 26455.321,E2 26455.321} C_VEL
LIN {X 0,Y 370.893,Z 998.664,A -85,B 0,C 180,E1 26460.014,E2 26460.014} C_VEL
LIN {X 0,Y 370.326,Z 1003.609,A -85,B 0,C 180,E1 26465.868,E2 26465.868} C_VEL
LIN {X 0,Y 370.252,Z 1010.975,A -85,B 0,C 180,E1 26470.597,E2 26470.597} C_VEL
LIN {X 0,Y 369.868,Z 1017.066,A -85,B 0,C 180,E1 26473.389,E2 26473.389} C_VEL
LIN {X 0,Y 341.811,Z 1056.572,A -85,B 0,C 180,E1 26476.797,E2 26476.797} C_VEL
LIN {X 0,Y 310.425,Z 1093.167,A -85,B 0,C 180,E1 26481.428,E2 26481.428} C_VEL
LIN {X 0,Y 280.188,Z 1124.018,A -85,B 0,C 180,E1 26487.427,E2 26487.427} C_VEL
LIN {X 0,Y 250.804,Z 1150.635,A -85,B 0,C 180,E1 26495.58,E2 26495.58} C_VEL
LIN {X 0,Y 227.006,Z 1171.338,A -85,B 0,C 180,E1 26505.654,E2 26505.654} C_VEL
LIN {X 0,Y 210.398,Z 1186.172,A -85,B 0,C 180,E1 26517.405,E2 26517.405} C_VEL
LIN {X 0,Y 201.412,Z 1196.201,A -85,B 0,C 180,E1 26530.714,E2 26530.714} C_VEL
LIN {X 0,Y 198.965,Z 1200.338,A -85,B 0,C 180,E1 26541.261,E2 26541.261} C_VEL
LIN {X 0,Y 199.222,Z 1201.555,A -85,B 0,C 180,E1 26549.998,E2 26549.998} C_VEL
LIN {X 0,Y 198.988,Z 1200.269,A -85,B 0,C 180,E1 26559.057,E2 26559.057} C_VEL
LIN {X 0,Y 201.407,Z 1196.225,A -85,B 0,C 180,E1 26569.283,E2 26569.283} C_VEL
LIN {X 0,Y 210.411,Z 1186.214,A -85,B 0,C 180,E1 26582.588,E2 26582.588} C_VEL
LIN {X 0,Y 228.754,Z 1169.856,A -85,B 0,C 180,E1 26595.243,E2 26595.243} C_VEL
LIN {X 0,Y 256.11,Z 1146.191,A -85,B 0,C 180,E1 26606.099,E2 26606.099} C_VEL
LIN {X 0,Y 285.021,Z 1119.388,A -85,B 0,C 180,E1 26613.65,E2 26613.65} C_VEL
LIN {X 0,Y 316.558,Z 1086.793,A -85,B 0,C 180,E1 26619.543,E2 26619.543} C_VEL
LIN {X 0,Y 346.242,Z 1050.952,A -85,B 0,C 180,E1 26623.766,E2 26623.766} C_VEL
LIN {X 0,Y 369.877,Z 1017.402,A -85,B 0,C 180,E1 26626.588,E2 26626.588} C_VEL
LIN {X 0,Y 370.41,Z 1007.647,A -85,B 0,C 180,E1 26631.434,E2 26631.434} C_VEL
LIN {X 0,Y 370.469,Z 1001.47,A -85,B 0,C 180,E1 26636.479,E2 26636.479} C_VEL
LIN {X 0,Y 371.021,Z 998.9,A -85,B 0,C 180,E1 26639.986,E2 26639.986} C_VEL
LIN {X 0,Y 369.286,Z 1003.064,A -85,B 0,C 180,E1 26645.857,E2 26645.857} C_VEL
LIN {X 0,Y 367.724,Z 1012.048,A -85,B 0,C 180,E1 26651.841,E2 26651.841} C_VEL
LIN {X 0,Y 366.827,Z 1017.852,A -85,B 0,C 180,E1 26654.491,E2 26654.491} C_VEL
LIN {X 0,Y 339.693,Z 1054.481,A -85,B 0,C 180,E1 26658.019,E2 26658.019} C_VEL
LIN {X 0,Y 309.297,Z 1088.886,A -85,B 0,C 180,E1 26662.733,E2 26662.733} C_VEL
LIN {X 0,Y 279.94,Z 1117.544,A -85,B 0,C 180,E1 26668.7,E2 26668.7} C_VEL
LIN {X 0,Y 271.035,Z 1125.643,A -85,B 0,C 180,E1 26670.913,E2 26670.913} C_VEL
LIN {X 0,Y 258.935,Z 1134.333,A -85,B 0,C 180,E1 26672.907,E2 26672.907} C_VEL
LIN {X 0,Y 246.819,Z 1142.407,A -85,B 0,C 180,E1 26675.127,E2 26675.127} C_VEL
LIN {X 0,Y 221.49,Z 1162.107,A -85,B 0,C 180,E1 26685.465,E2 26685.465} C_VEL
LIN {X 0,Y 202.82,Z 1176.67,A -85,B 0,C 180,E1 26698.567,E2 26698.567} C_VEL
LIN {X 0,Y 193.766,Z 1184.91,A -85,B 0,C 180,E1 26711.826,E2 26711.826} C_VEL
LIN {X 0,Y 191.024,Z 1188.436,A -85,B 0,C 180,E1 26725.465,E2 26725.465} C_VEL
LIN {X 0,Y 191.264,Z 1188.737,A -85,B 0,C 180,E1 26730.002,E2 26730.002} C_VEL
LIN {X 0,Y 191.379,Z 1187.671,A -85,B 0,C 180,E1 26739.088,E2 26739.088} C_VEL
LIN {X 0,Y 196.016,Z 1182.558,A -85,B 0,C 180,E1 26752.674,E2 26752.674} C_VEL
LIN {X 0,Y 207.67,Z 1172.825,A -85,B 0,C 180,E1 26765.602,E2 26765.602} C_VEL
LIN {X 0,Y 229.587,Z 1155.809,A -85,B 0,C 180,E1 26778.296,E2 26778.296} C_VEL
LIN {X 0,Y 255.618,Z 1135.214,A -85,B 0,C 180,E1 26787.512,E2 26787.512} C_VEL
LIN {X 0,Y 287.546,Z 1107.196,A -85,B 0,C 180,E1 26795.162,E2 26795.162} C_VEL
LIN {X 0,Y 317.99,Z 1076.615,A -85,B 0,C 180,E1 26800.478,E2 26800.478} C_VEL
LIN {X 0,Y 349.085,Z 1039.702,A -85,B 0,C 180,E1 26804.695,E2 26804.695} C_VEL
LIN {X 0,Y 361.778,Z 1022.445,A -85,B 0,C 180,E1 26806.209,E2 26806.209} C_VEL
LIN {X 0,Y 363.368,Z 1014.194,A -85,B 0,C 180,E1 26810.44,E2 26810.44} C_VEL
LIN {X 0,Y 364.792,Z 1008.225,A -85,B 0,C 180,E1 26815.262,E2 26815.262} C_VEL
LIN {X 0,Y 366.435,Z 1005.215,A -85,B 0,C 180,E1 26820.014,E2 26820.014} C_VEL
LIN {X 0,Y 365.696,Z 1010.245,A -85,B 0,C 180,E1 26825.943,E2 26825.943} C_VEL
LIN {X 0,Y 365.172,Z 1019.103,A -85,B 0,C 180,E1 26831.409,E2 26831.409} C_VEL
LIN {X 0,Y 365.014,Z 1021.126,A -85,B 0,C 180,E1 26832.337,E2 26832.337} C_VEL
LIN {X 0,Y 362.212,Z 1025.829,A -85,B 0,C 180,E1 26832.864,E2 26832.864} C_VEL
LIN {X 0,Y 333.085,Z 1064.1,A -85,B 0,C 180,E1 26836.305,E2 26836.305} C_VEL
LIN {X 0,Y 301.495,Z 1099.31,A -85,B 0,C 180,E1 26841.009,E2 26841.009} C_VEL
LIN {X 0,Y 268.728,Z 1130.664,A -85,B 0,C 180,E1 26847.665,E2 26847.665} C_VEL
LIN {X 0,Y 239.483,Z 1155.892,A -85,B 0,C 180,E1 26856.243,E2 26856.243} C_VEL
LIN {X 0,Y 215.468,Z 1175.623,A -85,B 0,C 180,E1 26867.283,E2 26867.283} C_VEL
LIN {X 0,Y 199.647,Z 1189.533,A -85,B 0,C 180,E1 26880.158,E2 26880.158} C_VEL
LIN {X 0,Y 193.055,Z 1196.933,A -85,B 0,C 180,E1 26891.752,E2 26891.752} C_VEL
LIN {X 0,Y 191.115,Z 1200.077,A -85,B 0,C 180,E1 26900.899,E2 26900.899} C_VEL
LIN {X 0,Y 191.329,Z 1201.296,A -85,B 0,C 180,E1 26909.998,E2 26909.998} C_VEL
LIN {X 0,Y 191.113,Z 1200.088,A -85,B 0,C 180,E1 26919.097,E2 26919.097} C_VEL
LIN {X 0,Y 194.035,Z 1195.562,A -85,B 0,C 180,E1 26930.793,E2 26930.793} C_VEL
LIN {X 0,Y 204.68,Z 1184.945,A -85,B 0,C 180,E1 26944.899,E2 26944.899} C_VEL
LIN {X 0,Y 222.983,Z 1169.584,A -85,B 0,C 180,E1 26956.758,E2 26956.758} C_VEL
LIN {X 0,Y 250.892,Z 1146.458,A -85,B 0,C 180,E1 26967.478,E2 26967.478} C_VEL
LIN {X 0,Y 280.696,Z 1119.822,A -85,B 0,C 180,E1 26975.01,E2 26975.01} C_VEL
LIN {X 0,Y 313.267,Z 1087.052,A -85,B 0,C 180,E1 26980.878,E2 26980.878} C_VEL
LIN {X 0,Y 343.231,Z 1051.737,A -85,B 0,C 180,E1 26984.978,E2 26984.978} C_VEL
LIN {X 0,Y 364.133,Z 1023.262,A -85,B 0,C 180,E1 26987.325,E2 26987.325} C_VEL
LIN {X 0,Y 365.081,Z 1020.584,A -85,B 0,C 180,E1 26988.043,E2 26988.043} C_VEL
LIN {X 0,Y 365.711,Z 1011.971,A -85,B 0,C 180,E1 26992.866,E2 26992.866} C_VEL
LIN {X 0,Y 366.112,Z 1007.064,A -85,B 0,C 180,E1 26997.621,E2 26997.621} C_VEL
LIN {X 0,Y 366.558,Z 1005.458,A -85,B 0,C 180,E1 26999.986,E2 26999.986} C_VEL
LIN {X 0,Y 364.589,Z 1009.588,A -85,B 0,C 180,E1 27005.899,E2 27005.899} C_VEL
LIN {X 0,Y 362.908,Z 1017.698,A -85,B 0,C 180,E1 27011.392,E2 27011.392} C_VEL
LIN {X 0,Y 362.135,Z 1021.954,A -85,B 0,C 180,E1 27013.484,E2 27013.484} C_VEL
LIN {X 0,Y 358.378,Z 1027.459,A -85,B 0,C 180,E1 27014.121,E2 27014.121} C_VEL
LIN {X 0,Y 329.292,Z 1064.239,A -85,B 0,C 180,E1 27017.789,E2 27017.789} C_VEL
LIN {X 0,Y 299.108,Z 1096.249,A -85,B 0,C 180,E1 27022.563,E2 27022.563} C_VEL
LIN {X 0,Y 267.511,Z 1125.347,A -85,B 0,C 180,E1 27029.227,E2 27029.227} C_VEL
LIN {X 0,Y 246.819,Z 1142.407,A -85,B 0,C 180,E1 27035.127,E2 27035.127} C_VEL
LIN {X 0,Y 234.974,Z 1149.94,A -85,B 0,C 180,E1 27037.624,E2 27037.624} C_VEL
LIN {X 0,Y 223.281,Z 1156.799,A -85,B 0,C 180,E1 27040.412,E2 27040.412} C_VEL
LIN {X 0,Y 200.936,Z 1173.224,A -85,B 0,C 180,E1 27053.016,E2 27053.016} C_VEL
LIN {X 0,Y 188.545,Z 1182.894,A -85,B 0,C 180,E1 27066.379,E2 27066.379} C_VEL
LIN {X 0,Y 183.499,Z 1187.963,A -85,B 0,C 180,E1 27080.523,E2 27080.523} C_VEL
LIN {X 0,Y 183.358,Z 1188.997,A -85,B 0,C 180,E1 27090.002,E2 27090.002} C_VEL
LIN {X 0,Y 183.518,Z 1187.932,A -85,B 0,C 180,E1 27099.481,E2 27099.481} C_VEL
LIN {X 0,Y 187.058,Z 1184.184,A -85,B 0,C 180,E1 27110.867,E2 27110.867} C_VEL
LIN {X 0,Y 198.426,Z 1174.975,A -85,B 0,C 180,E1 27124.834,E2 27124.834} C_VEL
LIN {X 0,Y 217.449,Z 1161.087,A -85,B 0,C 180,E1 27136.859,E2 27136.859} C_VEL
LIN {X 0,Y 243.673,Z 1141.402,A -85,B 0,C 180,E1 27146.848,E2 27146.848} C_VEL
LIN {X 0,Y 275.375,Z 1115.455,A -85,B 0,C 180,E1 27154.885,E2 27154.885} C_VEL
LIN {X 0,Y 308.859,Z 1083.628,A -85,B 0,C 180,E1 27160.891,E2 27160.891} C_VEL
LIN {X 0,Y 339.325,Z 1049.649,A -85,B 0,C 180,E1 27165.082,E2 27165.082} C_VEL
LIN {X 0,Y 356.627,Z 1027.262,A -85,B 0,C 180,E1 27167.055,E2 27167.055} C_VEL
LIN {X 0,Y 358.819,Z 1018.997,A -85,B 0,C 180,E1 27171.539,E2 27171.539} C_VEL
LIN {X 0,Y 360.849,Z 1012.748,A -85,B 0,C 180,E1 27177.614,E2 27177.614} C_VEL
LIN {X 0,Y 361.753,Z 1011.627,A -85,B 0,C 180,E1 27180.014,E2 27180.014} C_VEL
LIN {X 0,Y 360.861,Z 1016.738,A -85,B 0,C 180,E1 27186.022,E2 27186.022} C_VEL
LIN {X 0,Y 360.29,Z 1024.362,A -85,B 0,C 180,E1 27190.806,E2 27190.806} C_VEL
LIN {X 0,Y 359.397,Z 1027.049,A -85,B 0,C 180,E1 27191.708,E2 27191.708} C_VEL
LIN {X 0,Y 329.698,Z 1065.214,A -85,B 0,C 180,E1 27195.085,E2 27195.085} C_VEL
LIN {X 0,Y 298.006,Z 1099.63,A -85,B 0,C 180,E1 27199.626,E2 27199.626} C_VEL
LIN {X 0,Y 263.582,Z 1131.612,A -85,B 0,C 180,E1 27206.388,E2 27206.388} C_VEL
LIN {X 0,Y 234.852,Z 1155.457,A -85,B 0,C 180,E1 27214.528,E2 27214.528} C_VEL
LIN {X 0,Y 207.912,Z 1176.603,A -85,B 0,C 180,E1 27226.646,E2 27226.646} C_VEL
LIN {X 0,Y 191.394,Z 1190.253,A -85,B 0,C 180,E1 27240.323,E2 27240.323} C_VEL
LIN {X 0,Y 185.376,Z 1196.667,A -85,B 0,C 180,E1 27250.968,E2 27250.968} C_VEL
LIN {X 0,Y 183.06,Z 1200.219,A -85,B 0,C 180,E1 27262.273,E2 27262.273} C_VEL
